(* Logix 5000 project; controller reports 1756-L63 rev 20.15; software revision 20.04; part 39 of 52 *)

        [72].log_data[43].total := -975.3802, [72].log_data[43].time := 3600.0, [72].log_data[43].valid := 1, [72].log_data[44].min := -0.30000305, [72].log_data[44].max := -0.30000305, [72].log_data[44].total := -1080.0911, [72].log_data[44].time := 3600.0, [72].log_data[44].valid := 1, [72].log_data[45].time := 3600.0, [72].log_data[45].valid := 1, [72].log_data[46].time := 3600.0, [72].log_data[46].valid := 1, [72].log_data[47].time := 3600.0, [72].log_data[47].valid := 1, [72].log_data[48].min := 6.57968, [72].log_data[48].max := 6.8025494, [72].log_data[48].total := 24189.488, [72].log_data[48].time := 3600.0, [72].log_data[48].minminute := 18, [72].log_data[48].maxminute := 33, [72].log_data[48].valid := 1, [72].log_data[49].min := 7.0676346, [72].log_data[49].max := 9.6694765, [72].log_data[49].total := 30225.078, [72].log_data[49].time := 3600.0, [72].log_data[49].minminute := 14, [72].log_data[49].maxminute := 59, [72].log_data[49].valid := 1, [72].log_data[50].min := 2.124167, [72].log_data[50].max := 2.2044892, [72].log_data[50].total := 7798.3384, [72].log_data[50].time := 3600.0, [72].log_data[50].minminute := 59, [72].log_data[50].maxminute := 1, [72].log_data[50].valid := 1, [72].log_data[51].time := 3600.0, [72].log_data[51].valid := 1, [72].log_data[52].min := -2.9800034, [72].log_data[52].max := 0.11999512, [72].log_data[52].total := -7899.8555, [72].log_data[52].time := 3600.0, [72].log_data[52].minminute := 36, [72].log_data[52].maxminute := 3, [72].log_data[52].valid := 1, [72].log_data[53].min := -2.5800018, [72].log_data[53].max := 0.19999695, [72].log_data[53].total := -7610.7764, [72].log_data[53].time := 3600.0, [72].log_data[53].minminute := 55, [72].log_data[53].maxminute := 9, [72].log_data[53].valid := 1, [72].log_data[54].max := 0.523, [72].log_data[54].total := 1217.2916, [72].log_data[54].time := 3600.0, [72].log_data[54].minminute := 3, [72].log_data[54].maxminute := 57, [72].log_data[54].valid := 1, [72].log_data[55].max := 0.509, [72].log_data[55].total := 1254.1338, [72].log_data[55].time := 3600.0,
        [72].log_data[55].minminute := 7, [72].log_data[55].maxminute := 9, [72].log_data[55].valid := 1, [72].log_data[56].min := 0.16004932, [72].log_data[56].max := 0.16055967, [72].log_data[56].total := 576.9628, [72].log_data[56].time := 3600.0, [72].log_data[56].minminute := 16, [72].log_data[56].maxminute := 29, [72].log_data[56].valid := 1, [72].log_data[57].min := 0.2558395, [72].log_data[57].max := 0.25772393, [72].log_data[57].total := 923.43195, [72].log_data[57].time := 3600.0, [72].log_data[57].minminute := 27, [72].log_data[57].maxminute := 4, [72].log_data[57].valid := 1, [72].log_data[58].time := 3600.0, [72].log_data[58].valid := 1, [72].log_data[59].time := 3600.0, [72].log_data[59].valid := 1, [72].log_data[60].valid := 1, [72].log_data[61].valid := 1, [72].log_data[62].valid := 1, [72].log_data[63].valid := 1, [72].log_data[64].valid := 1, [72].log_data[65].valid := 1, [72].log_data[66].valid := 1, [72].log_data[67].valid := 1, [72].log_data[68].valid := 1, [72].log_data[69].valid := 1, [72].log_data[70].valid := 1, [72].log_data[71].valid := 1, [72].log_data[72].valid := 1, [72].log_data[73].valid := 1, [72].log_data[74].valid := 1, [72].log_data[75].valid := 1, [72].log_data[76].valid := 1, [72].log_data[77].valid := 1, [72].log_data[78].valid := 1, [72].log_data[79].valid := 1, [72].log_data[80].valid := 1, [72].log_data[81].valid := 1, [72].log_data[82].valid := 1, [72].log_data[83].valid := 1, [72].log_data[84].valid := 1, [72].log_data[85].valid := 1, [72].log_data[86].valid := 1, [72].log_data[87].valid := 1, [72].log_data[88].valid := 1, [72].log_data[89].valid := 1, [72].log_data[90].valid := 1, [72].log_data[91].valid := 1, [72].log_data[92].valid := 1, [72].log_data[93].valid := 1, [72].log_data[94].valid := 1, [72].log_data[95].valid := 1, [72].log_data[96].valid := 1, [72].log_data[97].valid := 1, [72].log_data[98].valid := 1,
        [72].log_data[99].valid := 1, [72].log_data[100].valid := 1, [72].log_data[101].valid := 1, [72].log_data[102].valid := 1, [72].log_data[103].valid := 1, [72].log_data[104].valid := 1, [72].log_data[105].valid := 1, [72].log_data[106].valid := 1, [72].log_data[107].valid := 1, [72].log_data[108].valid := 1, [72].log_data[109].valid := 1, [72].log_data[110].valid := 1, [72].log_data[111].valid := 1, [72].log_data[112].valid := 1, [72].log_data[113].valid := 1, [72].log_data[114].valid := 1, [72].log_data[115].valid := 1, [72].log_data[116].valid := 1, [72].log_data[117].valid := 1, [72].log_data[118].valid := 1, [72].log_data[119].valid := 1, [72].log_data[120].valid := 1, [72].log_data[121].valid := 1, [72].log_data[122].valid := 1, [72].log_data[123].valid := 1, [72].log_data[124].valid := 1, [72].time.Year := 2023, [72].time.Month := 1, [72].time.Day := 16, [72].time.Hour := 3, [72].time.Minute := 59, [72].time.Second := 59, [73].log_data[0].min := 1.0, [73].log_data[0].max := 1.0, [73].log_data[0].total := 3600.0, [73].log_data[0].time := 3600.0, [73].log_data[0].valid := 1, [73].log_data[1].time := 3600.0, [73].log_data[1].valid := 1, [73].log_data[2].time := 3600.0, [73].log_data[2].valid := 1, [73].log_data[3].time := 3600.0, [73].log_data[3].valid := 1, [73].log_data[4].time := 3600.0, [73].log_data[4].valid := 1, [73].log_data[5].time := 3600.0, [73].log_data[5].valid := 1, [73].log_data[6].time := 3600.0, [73].log_data[6].valid := 1, [73].log_data[7].time := 3600.0, [73].log_data[7].valid := 1, [73].log_data[8].min := 1.0, [73].log_data[8].max := 1.0, [73].log_data[8].total := 3600.0, [73].log_data[8].time := 3600.0, [73].log_data[8].valid := 1, [73].log_data[9].min := 1.0, [73].log_data[9].max := 1.0, [73].log_data[9].total := 3600.0, [73].log_data[9].time := 3600.0,
        [73].log_data[9].valid := 1, [73].log_data[10].min := 1.0, [73].log_data[10].max := 1.0, [73].log_data[10].total := 3600.0, [73].log_data[10].time := 3600.0, [73].log_data[10].valid := 1, [73].log_data[11].time := 3600.0, [73].log_data[11].valid := 1, [73].log_data[12].min := 1.0, [73].log_data[12].max := 1.0, [73].log_data[12].total := 3600.0, [73].log_data[12].time := 3600.0, [73].log_data[12].valid := 1, [73].log_data[13].min := 1.0, [73].log_data[13].max := 1.0, [73].log_data[13].total := 3600.0, [73].log_data[13].time := 3600.0, [73].log_data[13].valid := 1, [73].log_data[14].time := 3600.0, [73].log_data[14].valid := 1, [73].log_data[15].time := 3600.0, [73].log_data[15].valid := 1, [73].log_data[16].time := 3600.0, [73].log_data[16].valid := 1, [73].log_data[17].min := 1.0, [73].log_data[17].max := 1.0, [73].log_data[17].total := 3600.0, [73].log_data[17].time := 3600.0, [73].log_data[17].valid := 1, [73].log_data[18].time := 3600.0, [73].log_data[18].valid := 1, [73].log_data[19].time := 3600.0, [73].log_data[19].valid := 1, [73].log_data[20].time := 3600.0, [73].log_data[20].valid := 1, [73].log_data[21].min := 1.0, [73].log_data[21].max := 1.0, [73].log_data[21].total := 3600.0, [73].log_data[21].time := 3600.0, [73].log_data[21].valid := 1, [73].log_data[22].time := 3600.0, [73].log_data[22].valid := 1, [73].log_data[23].time := 3600.0, [73].log_data[23].valid := 1, [73].log_data[24].time := 3600.0, [73].log_data[24].valid := 1, [73].log_data[25].time := 3600.0, [73].log_data[25].valid := 1, [73].log_data[26].time := 3600.0, [73].log_data[26].valid := 1, [73].log_data[27].time := 3600.0, [73].log_data[27].valid := 1, [73].log_data[28].time := 3600.0, [73].log_data[28].valid := 1, [73].log_data[29].min := 1.0, [73].log_data[29].max := 1.0, [73].log_data[29].total := 3600.0, [73].log_data[29].time := 3600.0, [73].log_data[29].valid := 1, [73].log_data[30].min := 1.0,
        [73].log_data[30].max := 1.0, [73].log_data[30].total := 3600.0, [73].log_data[30].time := 3600.0, [73].log_data[30].valid := 1, [73].log_data[31].max := 1.0, [73].log_data[31].total := 1498.749, [73].log_data[31].time := 3600.0, [73].log_data[31].minminute := 6, [73].log_data[31].valid := 1, [73].log_data[32].max := 1.0, [73].log_data[32].total := 1630.249, [73].log_data[32].time := 3600.0, [73].log_data[32].maxminute := 8, [73].log_data[32].valid := 1, [73].log_data[33].time := 3600.0, [73].log_data[33].valid := 1, [73].log_data[34].time := 3600.0, [73].log_data[34].valid := 1, [73].log_data[35].max := 1.0, [73].log_data[35].total := 1629.998, [73].log_data[35].time := 3600.0, [73].log_data[35].maxminute := 1, [73].log_data[35].valid := 1, [73].log_data[36].max := 1.0, [73].log_data[36].total := 1440.7471, [73].log_data[36].time := 3600.0, [73].log_data[36].valid := 1, [73].log_data[37].time := 3600.0, [73].log_data[37].valid := 1, [73].log_data[38].time := 3600.0, [73].log_data[38].valid := 1, [73].log_data[39].min := 0.99635506, [73].log_data[39].max := 1.0070726, [73].log_data[39].total := 3607.0815, [73].log_data[39].time := 3600.0, [73].log_data[39].minminute := 25, [73].log_data[39].maxminute := 53, [73].log_data[39].valid := 1, [73].log_data[40].min := 7.584652, [73].log_data[40].max := 7.597843, [73].log_data[40].total := 27334.826, [73].log_data[40].time := 3600.0, [73].log_data[40].minminute := 3, [73].log_data[40].maxminute := 12, [73].log_data[40].valid := 1, [73].log_data[41].min := 0.022540038, [73].log_data[41].max := 0.03529907, [73].log_data[41].total := 104.06682, [73].log_data[41].time := 3600.0, [73].log_data[41].maxminute := 33, [73].log_data[41].valid := 1, [73].log_data[42].min := 2.2918782, [73].log_data[42].max := 2.2964714, [73].log_data[42].total := 8259.474, [73].log_data[42].time := 3600.0, [73].log_data[42].minminute := 2, [73].log_data[42].maxminute := 2, [73].log_data[42].valid := 1, [73].log_data[43].min := -0.27999878, [73].log_data[43].max := -0.26000214,
        [73].log_data[43].total := -978.1933, [73].log_data[43].time := 3600.0, [73].log_data[43].valid := 1, [73].log_data[44].min := -0.30000305, [73].log_data[44].max := -0.30000305, [73].log_data[44].total := -1080.0911, [73].log_data[44].time := 3600.0, [73].log_data[44].valid := 1, [73].log_data[45].time := 3600.0, [73].log_data[45].valid := 1, [73].log_data[46].time := 3600.0, [73].log_data[46].valid := 1, [73].log_data[47].time := 3600.0, [73].log_data[47].valid := 1, [73].log_data[48].min := 6.747862, [73].log_data[48].max := 6.764351, [73].log_data[48].total := 24322.072, [73].log_data[48].time := 3600.0, [73].log_data[48].minminute := 58, [73].log_data[48].valid := 1, [73].log_data[49].min := 9.655932, [73].log_data[49].max := 9.74073, [73].log_data[49].total := 34957.934, [73].log_data[49].time := 3600.0, [73].log_data[49].maxminute := 58, [73].log_data[49].valid := 1, [73].log_data[50].min := 2.0386624, [73].log_data[50].max := 2.1277, [73].log_data[50].total := 7504.0176, [73].log_data[50].time := 3600.0, [73].log_data[50].minminute := 59, [73].log_data[50].valid := 1, [73].log_data[51].time := 3600.0, [73].log_data[51].valid := 1, [73].log_data[52].min := -3.1200027, [73].log_data[52].max := 0.11999512, [73].log_data[52].total := -8078.232, [73].log_data[52].time := 3600.0, [73].log_data[52].minminute := 18, [73].log_data[52].maxminute := 6, [73].log_data[52].valid := 1, [73].log_data[53].min := -2.6399994, [73].log_data[53].max := 0.16000366, [73].log_data[53].total := -7426.6094, [73].log_data[53].time := 3600.0, [73].log_data[53].minminute := 23, [73].log_data[53].maxminute := 1, [73].log_data[53].valid := 1, [73].log_data[54].max := 0.5445, [73].log_data[54].total := 1242.5043, [73].log_data[54].time := 3600.0, [73].log_data[54].minminute := 6, [73].log_data[54].maxminute := 18, [73].log_data[54].valid := 1, [73].log_data[55].max := 0.554, [73].log_data[55].total := 1217.1788, [73].log_data[55].time := 3600.0, [73].log_data[55].maxminute := 23, [73].log_data[55].valid := 1, [73].log_data[56].min := 0.16008857,
        [73].log_data[56].max := 0.16055967, [73].log_data[56].total := 576.96655, [73].log_data[56].time := 3600.0, [73].log_data[56].maxminute := 26, [73].log_data[56].valid := 1, [73].log_data[57].min := 0.255761, [73].log_data[57].max := 0.25619283, [73].log_data[57].total := 921.46454, [73].log_data[57].time := 3600.0, [73].log_data[57].minminute := 11, [73].log_data[57].maxminute := 14, [73].log_data[57].valid := 1, [73].log_data[58].time := 3600.0, [73].log_data[58].valid := 1, [73].log_data[59].time := 3600.0, [73].log_data[59].valid := 1, [73].log_data[60].valid := 1, [73].log_data[61].valid := 1, [73].log_data[62].valid := 1, [73].log_data[63].valid := 1, [73].log_data[64].valid := 1, [73].log_data[65].valid := 1, [73].log_data[66].valid := 1, [73].log_data[67].valid := 1, [73].log_data[68].valid := 1, [73].log_data[69].valid := 1, [73].log_data[70].valid := 1, [73].log_data[71].valid := 1, [73].log_data[72].valid := 1, [73].log_data[73].valid := 1, [73].log_data[74].valid := 1, [73].log_data[75].valid := 1, [73].log_data[76].valid := 1, [73].log_data[77].valid := 1, [73].log_data[78].valid := 1, [73].log_data[79].valid := 1, [73].log_data[80].valid := 1, [73].log_data[81].valid := 1, [73].log_data[82].valid := 1, [73].log_data[83].valid := 1, [73].log_data[84].valid := 1, [73].log_data[85].valid := 1, [73].log_data[86].valid := 1, [73].log_data[87].valid := 1, [73].log_data[88].valid := 1, [73].log_data[89].valid := 1, [73].log_data[90].valid := 1, [73].log_data[91].valid := 1, [73].log_data[92].valid := 1, [73].log_data[93].valid := 1, [73].log_data[94].valid := 1, [73].log_data[95].valid := 1, [73].log_data[96].valid := 1, [73].log_data[97].valid := 1, [73].log_data[98].valid := 1, [73].log_data[99].valid := 1, [73].log_data[100].valid := 1, [73].log_data[101].valid := 1, [73].log_data[102].valid := 1, [73].log_data[103].valid := 1,
        [73].log_data[104].valid := 1, [73].log_data[105].valid := 1, [73].log_data[106].valid := 1, [73].log_data[107].valid := 1, [73].log_data[108].valid := 1, [73].log_data[109].valid := 1, [73].log_data[110].valid := 1, [73].log_data[111].valid := 1, [73].log_data[112].valid := 1, [73].log_data[113].valid := 1, [73].log_data[114].valid := 1, [73].log_data[115].valid := 1, [73].log_data[116].valid := 1, [73].log_data[117].valid := 1, [73].log_data[118].valid := 1, [73].log_data[119].valid := 1, [73].log_data[120].valid := 1, [73].log_data[121].valid := 1, [73].log_data[122].valid := 1, [73].log_data[123].valid := 1, [73].log_data[124].valid := 1, [73].time.Year := 2023, [73].time.Month := 1, [73].time.Day := 16, [73].time.Hour := 4, [73].time.Minute := 59, [73].time.Second := 59, [74].log_data[0].min := 1.0, [74].log_data[0].max := 1.0, [74].log_data[0].total := 3600.0, [74].log_data[0].time := 3600.0, [74].log_data[0].valid := 1, [74].log_data[1].time := 3600.0, [74].log_data[1].valid := 1, [74].log_data[2].time := 3600.0, [74].log_data[2].valid := 1, [74].log_data[3].time := 3600.0, [74].log_data[3].valid := 1, [74].log_data[4].time := 3600.0, [74].log_data[4].valid := 1, [74].log_data[5].time := 3600.0, [74].log_data[5].valid := 1, [74].log_data[6].time := 3600.0, [74].log_data[6].valid := 1, [74].log_data[7].time := 3600.0, [74].log_data[7].valid := 1, [74].log_data[8].max := 1.0, [74].log_data[8].total := 1742.751, [74].log_data[8].time := 3600.0, [74].log_data[8].minminute := 29, [74].log_data[8].valid := 1, [74].log_data[9].max := 1.0, [74].log_data[9].total := 1742.751, [74].log_data[9].time := 3600.0, [74].log_data[9].minminute := 29, [74].log_data[9].valid := 1, [74].log_data[10].min := 1.0, [74].log_data[10].max := 1.0, [74].log_data[10].total := 3600.0, [74].log_data[10].time := 3600.0,
        [74].log_data[10].valid := 1, [74].log_data[11].time := 3600.0, [74].log_data[11].valid := 1, [74].log_data[12].min := 1.0, [74].log_data[12].max := 1.0, [74].log_data[12].total := 3600.0, [74].log_data[12].time := 3600.0, [74].log_data[12].valid := 1, [74].log_data[13].min := 1.0, [74].log_data[13].max := 1.0, [74].log_data[13].total := 3600.0, [74].log_data[13].time := 3600.0, [74].log_data[13].valid := 1, [74].log_data[14].time := 3600.0, [74].log_data[14].valid := 1, [74].log_data[15].time := 3600.0, [74].log_data[15].valid := 1, [74].log_data[16].time := 3600.0, [74].log_data[16].valid := 1, [74].log_data[17].min := 1.0, [74].log_data[17].max := 1.0, [74].log_data[17].total := 3600.0, [74].log_data[17].time := 3600.0, [74].log_data[17].valid := 1, [74].log_data[18].time := 3600.0, [74].log_data[18].valid := 1, [74].log_data[19].time := 3600.0, [74].log_data[19].valid := 1, [74].log_data[20].time := 3600.0, [74].log_data[20].valid := 1, [74].log_data[21].min := 1.0, [74].log_data[21].max := 1.0, [74].log_data[21].total := 3600.0, [74].log_data[21].time := 3600.0, [74].log_data[21].valid := 1, [74].log_data[22].time := 3600.0, [74].log_data[22].valid := 1, [74].log_data[23].time := 3600.0, [74].log_data[23].valid := 1, [74].log_data[24].time := 3600.0, [74].log_data[24].valid := 1, [74].log_data[25].time := 3600.0, [74].log_data[25].valid := 1, [74].log_data[26].time := 3600.0, [74].log_data[26].valid := 1, [74].log_data[27].time := 3600.0, [74].log_data[27].valid := 1, [74].log_data[28].time := 3600.0, [74].log_data[28].valid := 1, [74].log_data[29].min := 1.0, [74].log_data[29].max := 1.0, [74].log_data[29].total := 3600.0, [74].log_data[29].time := 3600.0, [74].log_data[29].valid := 1, [74].log_data[30].min := 1.0, [74].log_data[30].max := 1.0, [74].log_data[30].total := 3600.0, [74].log_data[30].time := 3600.0, [74].log_data[30].valid := 1, [74].log_data[31].max := 1.0,
        [74].log_data[31].total := 968.99805, [74].log_data[31].time := 3600.0, [74].log_data[31].valid := 1, [74].log_data[32].max := 1.0, [74].log_data[32].total := 543.249, [74].log_data[32].time := 3600.0, [74].log_data[32].maxminute := 11, [74].log_data[32].valid := 1, [74].log_data[33].time := 3600.0, [74].log_data[33].valid := 1, [74].log_data[34].time := 3600.0, [74].log_data[34].valid := 1, [74].log_data[35].max := 1.0, [74].log_data[35].total := 724.749, [74].log_data[35].time := 3600.0, [74].log_data[35].maxminute := 5, [74].log_data[35].valid := 1, [74].log_data[36].max := 1.0, [74].log_data[36].total := 756.749, [74].log_data[36].time := 3600.0, [74].log_data[36].minminute := 3, [74].log_data[36].valid := 1, [74].log_data[37].time := 3600.0, [74].log_data[37].valid := 1, [74].log_data[38].time := 3600.0, [74].log_data[38].valid := 1, [74].log_data[39].min := 0.9936463, [74].log_data[39].max := 1.0061305, [74].log_data[39].total := 3601.6323, [74].log_data[39].time := 3600.0, [74].log_data[39].minminute := 3, [74].log_data[39].valid := 1, [74].log_data[40].min := 7.561569, [74].log_data[40].max := 7.609111, [74].log_data[40].total := 27332.018, [74].log_data[40].time := 3600.0, [74].log_data[40].minminute := 2, [74].log_data[40].maxminute := 4, [74].log_data[40].valid := 1, [74].log_data[41].min := 0.022540038, [74].log_data[41].max := 0.033139892, [74].log_data[41].total := 93.51873, [74].log_data[41].time := 3600.0, [74].log_data[41].minminute := 16, [74].log_data[41].valid := 1, [74].log_data[42].min := 2.2917604, [74].log_data[42].max := 2.2964714, [74].log_data[42].total := 8259.399, [74].log_data[42].time := 3600.0, [74].log_data[42].minminute := 17, [74].log_data[42].maxminute := 59, [74].log_data[42].valid := 1, [74].log_data[43].min := -0.27999878, [74].log_data[43].max := -0.26000214, [74].log_data[43].total := -968.6149, [74].log_data[43].time := 3600.0, [74].log_data[43].valid := 1, [74].log_data[44].min := -0.30000305, [74].log_data[44].max := -0.27999878, [74].log_data[44].total := -1080.0759,
        [74].log_data[44].time := 3600.0, [74].log_data[44].maxminute := 46, [74].log_data[44].valid := 1, [74].log_data[45].time := 3600.0, [74].log_data[45].valid := 1, [74].log_data[46].time := 3600.0, [74].log_data[46].valid := 1, [74].log_data[47].time := 3600.0, [74].log_data[47].valid := 1, [74].log_data[48].min := 6.734946, [74].log_data[48].max := 6.750061, [74].log_data[48].total := 24266.814, [74].log_data[48].time := 3600.0, [74].log_data[48].minminute := 35, [74].log_data[48].valid := 1, [74].log_data[49].min := 9.64867, [74].log_data[49].max := 9.741908, [74].log_data[49].total := 34884.496, [74].log_data[49].time := 3600.0, [74].log_data[49].minminute := 44, [74].log_data[49].maxminute := 8, [74].log_data[49].valid := 1, [74].log_data[50].min := 1.9993255, [74].log_data[50].max := 2.1042628, [74].log_data[50].total := 7410.9795, [74].log_data[50].time := 3600.0, [74].log_data[50].minminute := 29, [74].log_data[50].maxminute := 53, [74].log_data[50].valid := 1, [74].log_data[51].time := 3600.0, [74].log_data[51].valid := 1, [74].log_data[52].min := -3.0800018, [74].log_data[52].max := 0.11999512, [74].log_data[52].total := -6464.315, [74].log_data[52].time := 3600.0, [74].log_data[52].minminute := 1, [74].log_data[52].valid := 1, [74].log_data[53].min := -2.5800018, [74].log_data[53].max := 0.19999695, [74].log_data[53].total := -5924.441, [74].log_data[53].time := 3600.0, [74].log_data[53].minminute := 16, [74].log_data[53].maxminute := 4, [74].log_data[53].valid := 1, [74].log_data[54].max := 0.55050004, [74].log_data[54].total := 599.9697, [74].log_data[54].time := 3600.0, [74].log_data[54].maxminute := 22, [74].log_data[54].valid := 1, [74].log_data[55].max := 0.5245, [74].log_data[55].total := 587.57196, [74].log_data[55].time := 3600.0, [74].log_data[55].minminute := 3, [74].log_data[55].maxminute := 26, [74].log_data[55].valid := 1, [74].log_data[56].min := 0.16004932, [74].log_data[56].max := 0.16055967, [74].log_data[56].total := 576.99097, [74].log_data[56].time := 3600.0, [74].log_data[56].minminute := 23,
        [74].log_data[56].maxminute := 52, [74].log_data[56].valid := 1, [74].log_data[57].min := 0.25580025, [74].log_data[57].max := 0.25619283, [74].log_data[57].total := 921.4573, [74].log_data[57].time := 3600.0, [74].log_data[57].minminute := 4, [74].log_data[57].maxminute := 11, [74].log_data[57].valid := 1, [74].log_data[58].time := 3600.0, [74].log_data[58].valid := 1, [74].log_data[59].time := 3600.0, [74].log_data[59].valid := 1, [74].log_data[60].valid := 1, [74].log_data[61].valid := 1, [74].log_data[62].valid := 1, [74].log_data[63].valid := 1, [74].log_data[64].valid := 1, [74].log_data[65].valid := 1, [74].log_data[66].valid := 1, [74].log_data[67].valid := 1, [74].log_data[68].valid := 1, [74].log_data[69].valid := 1, [74].log_data[70].valid := 1, [74].log_data[71].valid := 1, [74].log_data[72].valid := 1, [74].log_data[73].valid := 1, [74].log_data[74].valid := 1, [74].log_data[75].valid := 1, [74].log_data[76].valid := 1, [74].log_data[77].valid := 1, [74].log_data[78].valid := 1, [74].log_data[79].valid := 1, [74].log_data[80].valid := 1, [74].log_data[81].valid := 1, [74].log_data[82].valid := 1, [74].log_data[83].valid := 1, [74].log_data[84].valid := 1, [74].log_data[85].valid := 1, [74].log_data[86].valid := 1, [74].log_data[87].valid := 1, [74].log_data[88].valid := 1, [74].log_data[89].valid := 1, [74].log_data[90].valid := 1, [74].log_data[91].valid := 1, [74].log_data[92].valid := 1, [74].log_data[93].valid := 1, [74].log_data[94].valid := 1, [74].log_data[95].valid := 1, [74].log_data[96].valid := 1, [74].log_data[97].valid := 1, [74].log_data[98].valid := 1, [74].log_data[99].valid := 1, [74].log_data[100].valid := 1, [74].log_data[101].valid := 1, [74].log_data[102].valid := 1, [74].log_data[103].valid := 1, [74].log_data[104].valid := 1, [74].log_data[105].valid := 1, [74].log_data[106].valid := 1,
        [74].log_data[107].valid := 1, [74].log_data[108].valid := 1, [74].log_data[109].valid := 1, [74].log_data[110].valid := 1, [74].log_data[111].valid := 1, [74].log_data[112].valid := 1, [74].log_data[113].valid := 1, [74].log_data[114].valid := 1, [74].log_data[115].valid := 1, [74].log_data[116].valid := 1, [74].log_data[117].valid := 1, [74].log_data[118].valid := 1, [74].log_data[119].valid := 1, [74].log_data[120].valid := 1, [74].log_data[121].valid := 1, [74].log_data[122].valid := 1, [74].log_data[123].valid := 1, [74].log_data[124].valid := 1, [74].time.Year := 2023, [74].time.Month := 1, [74].time.Day := 16, [74].time.Hour := 5, [74].time.Minute := 59, [74].time.Second := 59, [75].log_data[0].min := 1.0, [75].log_data[0].max := 1.0, [75].log_data[0].total := 3600.0, [75].log_data[0].time := 3600.0, [75].log_data[0].valid := 1, [75].log_data[1].time := 3600.0, [75].log_data[1].valid := 1, [75].log_data[2].time := 3600.0, [75].log_data[2].valid := 1, [75].log_data[3].time := 3600.0, [75].log_data[3].valid := 1, [75].log_data[4].time := 3600.0, [75].log_data[4].valid := 1, [75].log_data[5].time := 3600.0, [75].log_data[5].valid := 1, [75].log_data[6].time := 3600.0, [75].log_data[6].valid := 1, [75].log_data[7].time := 3600.0, [75].log_data[7].valid := 1, [75].log_data[8].time := 3600.0, [75].log_data[8].valid := 1, [75].log_data[9].time := 3600.0, [75].log_data[9].valid := 1, [75].log_data[10].min := 1.0, [75].log_data[10].max := 1.0, [75].log_data[10].total := 3600.0, [75].log_data[10].time := 3600.0, [75].log_data[10].valid := 1, [75].log_data[11].time := 3600.0, [75].log_data[11].valid := 1, [75].log_data[12].min := 1.0, [75].log_data[12].max := 1.0, [75].log_data[12].total := 3600.0, [75].log_data[12].time := 3600.0, [75].log_data[12].valid := 1, [75].log_data[13].min := 1.0,
        [75].log_data[13].max := 1.0, [75].log_data[13].total := 3600.0, [75].log_data[13].time := 3600.0, [75].log_data[13].valid := 1, [75].log_data[14].time := 3600.0, [75].log_data[14].valid := 1, [75].log_data[15].time := 3600.0, [75].log_data[15].valid := 1, [75].log_data[16].time := 3600.0, [75].log_data[16].valid := 1, [75].log_data[17].min := 1.0, [75].log_data[17].max := 1.0, [75].log_data[17].total := 3600.0, [75].log_data[17].time := 3600.0, [75].log_data[17].valid := 1, [75].log_data[18].time := 3600.0, [75].log_data[18].valid := 1, [75].log_data[19].time := 3600.0, [75].log_data[19].valid := 1, [75].log_data[20].time := 3600.0, [75].log_data[20].valid := 1, [75].log_data[21].min := 1.0, [75].log_data[21].max := 1.0, [75].log_data[21].total := 3600.0, [75].log_data[21].time := 3600.0, [75].log_data[21].valid := 1, [75].log_data[22].time := 3600.0, [75].log_data[22].valid := 1, [75].log_data[23].time := 3600.0, [75].log_data[23].valid := 1, [75].log_data[24].time := 3600.0, [75].log_data[24].valid := 1, [75].log_data[25].time := 3600.0, [75].log_data[25].valid := 1, [75].log_data[26].time := 3600.0, [75].log_data[26].valid := 1, [75].log_data[27].time := 3600.0, [75].log_data[27].valid := 1, [75].log_data[28].time := 3600.0, [75].log_data[28].valid := 1, [75].log_data[29].min := 1.0, [75].log_data[29].max := 1.0, [75].log_data[29].total := 3600.0, [75].log_data[29].time := 3600.0, [75].log_data[29].valid := 1, [75].log_data[30].min := 1.0, [75].log_data[30].max := 1.0, [75].log_data[30].total := 3600.0, [75].log_data[30].time := 3600.0, [75].log_data[30].valid := 1, [75].log_data[31].time := 3600.0, [75].log_data[31].valid := 1, [75].log_data[32].time := 3600.0, [75].log_data[32].valid := 1, [75].log_data[33].time := 3600.0, [75].log_data[33].valid := 1, [75].log_data[34].time := 3600.0, [75].log_data[34].valid := 1, [75].log_data[35].time := 3600.0, [75].log_data[35].valid := 1,
        [75].log_data[36].time := 3600.0, [75].log_data[36].valid := 1, [75].log_data[37].time := 3600.0, [75].log_data[37].valid := 1, [75].log_data[38].time := 3600.0, [75].log_data[38].valid := 1, [75].log_data[39].min := 0.9941174, [75].log_data[39].max := 1.0055416, [75].log_data[39].total := 3601.261, [75].log_data[39].time := 3600.0, [75].log_data[39].minminute := 36, [75].log_data[39].maxminute := 43, [75].log_data[39].valid := 1, [75].log_data[40].min := 7.574485, [75].log_data[40].max := 7.6107597, [75].log_data[40].total := 27331.771, [75].log_data[40].time := 3600.0, [75].log_data[40].minminute := 34, [75].log_data[40].maxminute := 32, [75].log_data[40].valid := 1, [75].log_data[41].min := 0.022540038, [75].log_data[41].max := 0.039224852, [75].log_data[41].total := 90.41001, [75].log_data[41].time := 3600.0, [75].log_data[41].maxminute := 5, [75].log_data[41].valid := 1, [75].log_data[42].min := 2.2917604, [75].log_data[42].max := 2.2963536, [75].log_data[42].total := 8259.333, [75].log_data[42].time := 3600.0, [75].log_data[42].minminute := 3, [75].log_data[42].maxminute := 10, [75].log_data[42].valid := 1, [75].log_data[43].min := -0.27999878, [75].log_data[43].max := -0.26000214, [75].log_data[43].total := -959.8148, [75].log_data[43].time := 3600.0, [75].log_data[43].valid := 1, [75].log_data[44].min := -0.30000305, [75].log_data[44].max := -0.30000305, [75].log_data[44].total := -1080.0911, [75].log_data[44].time := 3600.0, [75].log_data[44].valid := 1, [75].log_data[45].time := 3600.0, [75].log_data[45].valid := 1, [75].log_data[46].time := 3600.0, [75].log_data[46].valid := 1, [75].log_data[47].time := 3600.0, [75].log_data[47].valid := 1, [75].log_data[48].min := 6.7382436, [75].log_data[48].max := 6.7473125, [75].log_data[48].total := 24275.645, [75].log_data[48].time := 3600.0, [75].log_data[48].maxminute := 48, [75].log_data[48].valid := 1, [75].log_data[49].min := 9.64553, [75].log_data[49].max := 9.706968, [75].log_data[49].total := 34838.707, [75].log_data[49].time := 3600.0, [75].log_data[49].minminute := 5,
        [75].log_data[49].maxminute := 48, [75].log_data[49].valid := 1, [75].log_data[50].min := 2.0994341, [75].log_data[50].max := 2.1086206, [75].log_data[50].total := 7579.887, [75].log_data[50].time := 3600.0, [75].log_data[50].maxminute := 44, [75].log_data[50].valid := 1, [75].log_data[51].time := 3600.0, [75].log_data[51].valid := 1, [75].log_data[52].min := -1.5999985, [75].log_data[52].max := -1.4400024, [75].log_data[52].total := -5502.215, [75].log_data[52].time := 3600.0, [75].log_data[52].minminute := 51, [75].log_data[52].maxminute := 15, [75].log_data[52].valid := 1, [75].log_data[53].min := -1.4400024, [75].log_data[53].max := -1.2399979, [75].log_data[53].total := -4781.3306, [75].log_data[53].time := 3600.0, [75].log_data[53].minminute := 7, [75].log_data[53].maxminute := 54, [75].log_data[53].valid := 1, [75].log_data[54].time := 3600.0, [75].log_data[54].valid := 1, [75].log_data[55].time := 3600.0, [75].log_data[55].valid := 1, [75].log_data[56].min := 0.16004932, [75].log_data[56].max := 0.16055967, [75].log_data[56].total := 576.94586, [75].log_data[56].time := 3600.0, [75].log_data[56].minminute := 8, [75].log_data[56].maxminute := 13, [75].log_data[56].valid := 1, [75].log_data[57].min := 0.25580025, [75].log_data[57].max := 0.25627133, [75].log_data[57].total := 921.7233, [75].log_data[57].time := 3600.0, [75].log_data[57].minminute := 24, [75].log_data[57].maxminute := 32, [75].log_data[57].valid := 1, [75].log_data[58].time := 3600.0, [75].log_data[58].valid := 1, [75].log_data[59].time := 3600.0, [75].log_data[59].valid := 1, [75].log_data[60].valid := 1, [75].log_data[61].valid := 1, [75].log_data[62].valid := 1, [75].log_data[63].valid := 1, [75].log_data[64].valid := 1, [75].log_data[65].valid := 1, [75].log_data[66].valid := 1, [75].log_data[67].valid := 1, [75].log_data[68].valid := 1, [75].log_data[69].valid := 1, [75].log_data[70].valid := 1, [75].log_data[71].valid := 1, [75].log_data[72].valid := 1, [75].log_data[73].valid := 1,
        [75].log_data[74].valid := 1, [75].log_data[75].valid := 1, [75].log_data[76].valid := 1, [75].log_data[77].valid := 1, [75].log_data[78].valid := 1, [75].log_data[79].valid := 1, [75].log_data[80].valid := 1, [75].log_data[81].valid := 1, [75].log_data[82].valid := 1, [75].log_data[83].valid := 1, [75].log_data[84].valid := 1, [75].log_data[85].valid := 1, [75].log_data[86].valid := 1, [75].log_data[87].valid := 1, [75].log_data[88].valid := 1, [75].log_data[89].valid := 1, [75].log_data[90].valid := 1, [75].log_data[91].valid := 1, [75].log_data[92].valid := 1, [75].log_data[93].valid := 1, [75].log_data[94].valid := 1, [75].log_data[95].valid := 1, [75].log_data[96].valid := 1, [75].log_data[97].valid := 1, [75].log_data[98].valid := 1, [75].log_data[99].valid := 1, [75].log_data[100].valid := 1, [75].log_data[101].valid := 1, [75].log_data[102].valid := 1, [75].log_data[103].valid := 1, [75].log_data[104].valid := 1, [75].log_data[105].valid := 1, [75].log_data[106].valid := 1, [75].log_data[107].valid := 1, [75].log_data[108].valid := 1, [75].log_data[109].valid := 1, [75].log_data[110].valid := 1, [75].log_data[111].valid := 1, [75].log_data[112].valid := 1, [75].log_data[113].valid := 1, [75].log_data[114].valid := 1, [75].log_data[115].valid := 1, [75].log_data[116].valid := 1, [75].log_data[117].valid := 1, [75].log_data[118].valid := 1, [75].log_data[119].valid := 1, [75].log_data[120].valid := 1, [75].log_data[121].valid := 1, [75].log_data[122].valid := 1, [75].log_data[123].valid := 1, [75].log_data[124].valid := 1, [75].time.Year := 2023, [75].time.Month := 1, [75].time.Day := 16, [75].time.Hour := 6, [75].time.Minute := 59, [75].time.Second := 59, [76].log_data[0].min := 1.0, [76].log_data[0].max := 1.0, [76].log_data[0].total := 3600.0,
        [76].log_data[0].time := 3600.0, [76].log_data[0].valid := 1, [76].log_data[1].max := 1.0, [76].log_data[1].total := 546.5, [76].log_data[1].time := 3600.0, [76].log_data[1].maxminute := 36, [76].log_data[1].valid := 1, [76].log_data[2].max := 1.0, [76].log_data[2].total := 543.0, [76].log_data[2].time := 3600.0, [76].log_data[2].maxminute := 36, [76].log_data[2].valid := 1, [76].log_data[3].time := 3600.0, [76].log_data[3].valid := 1, [76].log_data[4].time := 3600.0, [76].log_data[4].valid := 1, [76].log_data[5].max := 1.0, [76].log_data[5].total := 227.5, [76].log_data[5].time := 3600.0, [76].log_data[5].maxminute := 38, [76].log_data[5].valid := 1, [76].log_data[6].time := 3600.0, [76].log_data[6].valid := 1, [76].log_data[7].time := 3600.0, [76].log_data[7].valid := 1, [76].log_data[8].max := 1.0, [76].log_data[8].total := 1171.249, [76].log_data[8].time := 3600.0, [76].log_data[8].maxminute := 40, [76].log_data[8].valid := 1, [76].log_data[9].max := 1.0, [76].log_data[9].total := 1167.749, [76].log_data[9].time := 3600.0, [76].log_data[9].maxminute := 40, [76].log_data[9].valid := 1, [76].log_data[10].min := 1.0, [76].log_data[10].max := 1.0, [76].log_data[10].total := 3600.0, [76].log_data[10].time := 3600.0, [76].log_data[10].valid := 1, [76].log_data[11].time := 3600.0, [76].log_data[11].valid := 1, [76].log_data[12].min := 1.0, [76].log_data[12].max := 1.0, [76].log_data[12].total := 3600.0, [76].log_data[12].time := 3600.0, [76].log_data[12].valid := 1, [76].log_data[13].min := 1.0, [76].log_data[13].max := 1.0, [76].log_data[13].total := 3600.0, [76].log_data[13].time := 3600.0, [76].log_data[13].valid := 1, [76].log_data[14].time := 3600.0, [76].log_data[14].valid := 1, [76].log_data[15].time := 3600.0, [76].log_data[15].valid := 1, [76].log_data[16].time := 3600.0, [76].log_data[16].valid := 1, [76].log_data[17].min := 1.0, [76].log_data[17].max := 1.0,
        [76].log_data[17].total := 3600.0, [76].log_data[17].time := 3600.0, [76].log_data[17].valid := 1, [76].log_data[18].time := 3600.0, [76].log_data[18].valid := 1, [76].log_data[19].time := 3600.0, [76].log_data[19].valid := 1, [76].log_data[20].time := 3600.0, [76].log_data[20].valid := 1, [76].log_data[21].min := 1.0, [76].log_data[21].max := 1.0, [76].log_data[21].total := 3600.0, [76].log_data[21].time := 3600.0, [76].log_data[21].valid := 1, [76].log_data[22].time := 3600.0, [76].log_data[22].valid := 1, [76].log_data[23].time := 3600.0, [76].log_data[23].valid := 1, [76].log_data[24].time := 3600.0, [76].log_data[24].valid := 1, [76].log_data[25].time := 3600.0, [76].log_data[25].valid := 1, [76].log_data[26].time := 3600.0, [76].log_data[26].valid := 1, [76].log_data[27].time := 3600.0, [76].log_data[27].valid := 1, [76].log_data[28].time := 3600.0, [76].log_data[28].valid := 1, [76].log_data[29].min := 1.0, [76].log_data[29].max := 1.0, [76].log_data[29].total := 3600.0, [76].log_data[29].time := 3600.0, [76].log_data[29].valid := 1, [76].log_data[30].min := 1.0, [76].log_data[30].max := 1.0, [76].log_data[30].total := 3600.0, [76].log_data[30].time := 3600.0, [76].log_data[30].valid := 1, [76].log_data[31].max := 1.0, [76].log_data[31].total := 543.249, [76].log_data[31].time := 3600.0, [76].log_data[31].maxminute := 44, [76].log_data[31].valid := 1, [76].log_data[32].max := 1.0, [76].log_data[32].total := 444.498, [76].log_data[32].time := 3600.0, [76].log_data[32].maxminute := 40, [76].log_data[32].valid := 1, [76].log_data[33].time := 3600.0, [76].log_data[33].valid := 1, [76].log_data[34].time := 3600.0, [76].log_data[34].valid := 1, [76].log_data[35].max := 1.0, [76].log_data[35].total := 543.249, [76].log_data[35].time := 3600.0, [76].log_data[35].maxminute := 48, [76].log_data[35].valid := 1, [76].log_data[36].max := 1.0, [76].log_data[36].total := 440.998, [76].log_data[36].time := 3600.0,
        [76].log_data[36].maxminute := 40, [76].log_data[36].valid := 1, [76].log_data[37].max := 7.3416233, [76].log_data[37].total := 3478.435, [76].log_data[37].time := 3600.0, [76].log_data[37].maxminute := 38, [76].log_data[37].valid := 1, [76].log_data[38].time := 3600.0, [76].log_data[38].valid := 1, [76].log_data[39].min := 0.99435294, [76].log_data[39].max := 1.0215589, [76].log_data[39].total := 3607.7969, [76].log_data[39].time := 3600.0, [76].log_data[39].minminute := 14, [76].log_data[39].maxminute := 43, [76].log_data[39].valid := 1, [76].log_data[40].min := 7.584652, [76].log_data[40].max := 7.6019654, [76].log_data[40].total := 27338.77, [76].log_data[40].time := 3600.0, [76].log_data[40].minminute := 29, [76].log_data[40].maxminute := 5, [76].log_data[40].valid := 1, [76].log_data[41].min := 0.022540038, [76].log_data[41].max := 0.037261963, [76].log_data[41].total := 114.78345, [76].log_data[41].time := 3600.0, [76].log_data[41].maxminute := 41, [76].log_data[41].valid := 1, [76].log_data[42].min := 2.2917604, [76].log_data[42].max := 2.2964714, [76].log_data[42].total := 8259.297, [76].log_data[42].time := 3600.0, [76].log_data[42].minminute := 52, [76].log_data[42].maxminute := 20, [76].log_data[42].valid := 1, [76].log_data[43].min := -0.27999878, [76].log_data[43].max := -0.26000214, [76].log_data[43].total := -980.99854, [76].log_data[43].time := 3600.0, [76].log_data[43].valid := 1, [76].log_data[44].min := -0.30000305, [76].log_data[44].max := -0.30000305, [76].log_data[44].total := -1080.0911, [76].log_data[44].time := 3600.0, [76].log_data[44].valid := 1, [76].log_data[45].time := 3600.0, [76].log_data[45].valid := 1, [76].log_data[46].time := 3600.0, [76].log_data[46].valid := 1, [76].log_data[47].time := 3600.0, [76].log_data[47].valid := 1, [76].log_data[48].min := 6.6335416, [76].log_data[48].max := 6.9465485, [76].log_data[48].total := 24319.84, [76].log_data[48].time := 3600.0, [76].log_data[48].minminute := 59, [76].log_data[48].maxminute := 45, [76].log_data[48].valid := 1, [76].log_data[49].min := 7.204253,
        [76].log_data[49].max := 9.739357, [76].log_data[49].total := 33188.277, [76].log_data[49].time := 3600.0, [76].log_data[49].minminute := 59, [76].log_data[49].maxminute := 28, [76].log_data[49].valid := 1, [76].log_data[50].min := 2.061864, [76].log_data[50].max := 2.1505485, [76].log_data[50].total := 7572.1, [76].log_data[50].time := 3600.0, [76].log_data[50].minminute := 43, [76].log_data[50].maxminute := 40, [76].log_data[50].valid := 1, [76].log_data[51].time := 3600.0, [76].log_data[51].valid := 1, [76].log_data[52].min := -4.199997, [76].log_data[52].max := 0.11999512, [76].log_data[52].total := -6285.726, [76].log_data[52].time := 3600.0, [76].log_data[52].minminute := 40, [76].log_data[52].maxminute := 42, [76].log_data[52].valid := 1, [76].log_data[53].min := -3.9399948, [76].log_data[53].max := 0.27999878, [76].log_data[53].total := -5460.3057, [76].log_data[53].time := 3600.0, [76].log_data[53].minminute := 40, [76].log_data[53].maxminute := 58, [76].log_data[53].valid := 1, [76].log_data[54].max := 0.5535, [76].log_data[54].total := 389.23734, [76].log_data[54].time := 3600.0, [76].log_data[54].maxminute := 54, [76].log_data[54].valid := 1, [76].log_data[55].max := 0.5175, [76].log_data[55].total := 387.67783, [76].log_data[55].time := 3600.0, [76].log_data[55].maxminute := 40, [76].log_data[55].valid := 1, [76].log_data[56].min := 0.16008857, [76].log_data[56].max := 0.16048115, [76].log_data[56].total := 576.83215, [76].log_data[56].time := 3600.0, [76].log_data[56].minminute := 40, [76].log_data[56].maxminute := 14, [76].log_data[56].valid := 1, [76].log_data[57].min := 0.2558395, [76].log_data[57].max := 0.25627133, [76].log_data[57].total := 921.702, [76].log_data[57].time := 3600.0, [76].log_data[57].minminute := 41, [76].log_data[57].valid := 1, [76].log_data[58].time := 3600.0, [76].log_data[58].valid := 1, [76].log_data[59].time := 3600.0, [76].log_data[59].valid := 1, [76].log_data[60].valid := 1, [76].log_data[61].valid := 1, [76].log_data[62].valid := 1, [76].log_data[63].valid := 1,
        [76].log_data[64].valid := 1, [76].log_data[65].valid := 1, [76].log_data[66].valid := 1, [76].log_data[67].valid := 1, [76].log_data[68].valid := 1, [76].log_data[69].valid := 1, [76].log_data[70].valid := 1, [76].log_data[71].valid := 1, [76].log_data[72].valid := 1, [76].log_data[73].valid := 1, [76].log_data[74].valid := 1, [76].log_data[75].valid := 1, [76].log_data[76].valid := 1, [76].log_data[77].valid := 1, [76].log_data[78].valid := 1, [76].log_data[79].valid := 1, [76].log_data[80].valid := 1, [76].log_data[81].valid := 1, [76].log_data[82].valid := 1, [76].log_data[83].valid := 1, [76].log_data[84].valid := 1, [76].log_data[85].valid := 1, [76].log_data[86].valid := 1, [76].log_data[87].valid := 1, [76].log_data[88].valid := 1, [76].log_data[89].valid := 1, [76].log_data[90].valid := 1, [76].log_data[91].valid := 1, [76].log_data[92].valid := 1, [76].log_data[93].valid := 1, [76].log_data[94].valid := 1, [76].log_data[95].valid := 1, [76].log_data[96].valid := 1, [76].log_data[97].valid := 1, [76].log_data[98].valid := 1, [76].log_data[99].valid := 1, [76].log_data[100].valid := 1, [76].log_data[101].valid := 1, [76].log_data[102].valid := 1, [76].log_data[103].valid := 1, [76].log_data[104].valid := 1, [76].log_data[105].valid := 1, [76].log_data[106].valid := 1, [76].log_data[107].valid := 1, [76].log_data[108].valid := 1, [76].log_data[109].valid := 1, [76].log_data[110].valid := 1, [76].log_data[111].valid := 1, [76].log_data[112].valid := 1, [76].log_data[113].valid := 1, [76].log_data[114].valid := 1, [76].log_data[115].valid := 1, [76].log_data[116].valid := 1, [76].log_data[117].valid := 1, [76].log_data[118].valid := 1, [76].log_data[119].valid := 1, [76].log_data[120].valid := 1, [76].log_data[121].valid := 1, [76].log_data[122].valid := 1, [76].log_data[123].valid := 1,
        [76].log_data[124].valid := 1, [76].time.Year := 2023, [76].time.Month := 1, [76].time.Day := 16, [76].time.Hour := 7, [76].time.Minute := 59, [76].time.Second := 59, [77].log_data[0].min := 1.0, [77].log_data[0].max := 1.0, [77].log_data[0].total := 3600.0, [77].log_data[0].time := 3600.0, [77].log_data[0].valid := 1, [77].log_data[1].time := 3600.0, [77].log_data[1].valid := 1, [77].log_data[2].time := 3600.0, [77].log_data[2].valid := 1, [77].log_data[3].time := 3600.0, [77].log_data[3].valid := 1, [77].log_data[4].time := 3600.0, [77].log_data[4].valid := 1, [77].log_data[5].time := 3600.0, [77].log_data[5].valid := 1, [77].log_data[6].time := 3600.0, [77].log_data[6].valid := 1, [77].log_data[7].time := 3600.0, [77].log_data[7].valid := 1, [77].log_data[8].max := 1.0, [77].log_data[8].total := 3315.751, [77].log_data[8].time := 3600.0, [77].log_data[8].minminute := 55, [77].log_data[8].valid := 1, [77].log_data[9].max := 1.0, [77].log_data[9].total := 3315.751, [77].log_data[9].time := 3600.0, [77].log_data[9].minminute := 55, [77].log_data[9].valid := 1, [77].log_data[10].min := 1.0, [77].log_data[10].max := 1.0, [77].log_data[10].total := 3600.0, [77].log_data[10].time := 3600.0, [77].log_data[10].valid := 1, [77].log_data[11].time := 3600.0, [77].log_data[11].valid := 1, [77].log_data[12].min := 1.0, [77].log_data[12].max := 1.0, [77].log_data[12].total := 3600.0, [77].log_data[12].time := 3600.0, [77].log_data[12].valid := 1, [77].log_data[13].min := 1.0, [77].log_data[13].max := 1.0, [77].log_data[13].total := 3600.0, [77].log_data[13].time := 3600.0, [77].log_data[13].valid := 1, [77].log_data[14].time := 3600.0, [77].log_data[14].valid := 1, [77].log_data[15].time := 3600.0, [77].log_data[15].valid := 1, [77].log_data[16].time := 3600.0, [77].log_data[16].valid := 1, [77].log_data[17].min := 1.0,
        [77].log_data[17].max := 1.0, [77].log_data[17].total := 3600.0, [77].log_data[17].time := 3600.0, [77].log_data[17].valid := 1, [77].log_data[18].time := 3600.0, [77].log_data[18].valid := 1, [77].log_data[19].time := 3600.0, [77].log_data[19].valid := 1, [77].log_data[20].time := 3600.0, [77].log_data[20].valid := 1, [77].log_data[21].min := 1.0, [77].log_data[21].max := 1.0, [77].log_data[21].total := 3600.0, [77].log_data[21].time := 3600.0, [77].log_data[21].valid := 1, [77].log_data[22].time := 3600.0, [77].log_data[22].valid := 1, [77].log_data[23].time := 3600.0, [77].log_data[23].valid := 1, [77].log_data[24].time := 3600.0, [77].log_data[24].valid := 1, [77].log_data[25].time := 3600.0, [77].log_data[25].valid := 1, [77].log_data[26].time := 3600.0, [77].log_data[26].valid := 1, [77].log_data[27].time := 3600.0, [77].log_data[27].valid := 1, [77].log_data[28].time := 3600.0, [77].log_data[28].valid := 1, [77].log_data[29].min := 1.0, [77].log_data[29].max := 1.0, [77].log_data[29].total := 3600.0, [77].log_data[29].time := 3600.0, [77].log_data[29].valid := 1, [77].log_data[30].min := 1.0, [77].log_data[30].max := 1.0, [77].log_data[30].total := 3600.0, [77].log_data[30].time := 3600.0, [77].log_data[30].valid := 1, [77].log_data[31].max := 1.0, [77].log_data[31].total := 1575.2471, [77].log_data[31].time := 3600.0, [77].log_data[31].maxminute := 5, [77].log_data[31].valid := 1, [77].log_data[32].max := 1.0, [77].log_data[32].total := 1303.0, [77].log_data[32].time := 3600.0, [77].log_data[32].minminute := 3, [77].log_data[32].valid := 1, [77].log_data[33].time := 3600.0, [77].log_data[33].valid := 1, [77].log_data[34].time := 3600.0, [77].log_data[34].valid := 1, [77].log_data[35].max := 1.0, [77].log_data[35].total := 1328.2471, [77].log_data[35].time := 3600.0, [77].log_data[35].maxminute := 9, [77].log_data[35].valid := 1, [77].log_data[36].max := 1.0, [77].log_data[36].total := 1549.998,
        [77].log_data[36].time := 3600.0, [77].log_data[36].minminute := 7, [77].log_data[36].valid := 1, [77].log_data[37].time := 3600.0, [77].log_data[37].valid := 1, [77].log_data[38].time := 3600.0, [77].log_data[38].valid := 1, [77].log_data[39].min := 0.9956484, [77].log_data[39].max := 1.0080148, [77].log_data[39].total := 3607.7026, [77].log_data[39].time := 3600.0, [77].log_data[39].minminute := 44, [77].log_data[39].maxminute := 40, [77].log_data[39].valid := 1, [77].log_data[40].min := 7.5742097, [77].log_data[40].max := 7.609111, [77].log_data[40].total := 27335.467, [77].log_data[40].time := 3600.0, [77].log_data[40].minminute := 28, [77].log_data[40].maxminute := 24, [77].log_data[40].valid := 1, [77].log_data[41].min := 0.022540038, [77].log_data[41].max := 0.033139892, [77].log_data[41].total := 100.900345, [77].log_data[41].time := 3600.0, [77].log_data[41].minminute := 41, [77].log_data[41].maxminute := 16, [77].log_data[41].valid := 1, [77].log_data[42].min := 2.2916427, [77].log_data[42].max := 2.2963536, [77].log_data[42].total := 8259.254, [77].log_data[42].time := 3600.0, [77].log_data[42].minminute := 14, [77].log_data[42].maxminute := 39, [77].log_data[42].valid := 1, [77].log_data[43].min := -0.27999878, [77].log_data[43].max := -0.26000214, [77].log_data[43].total := -989.81494, [77].log_data[43].time := 3600.0, [77].log_data[43].valid := 1, [77].log_data[44].min := -0.3199997, [77].log_data[44].max := -0.30000305, [77].log_data[44].total := -1080.0961, [77].log_data[44].time := 3600.0, [77].log_data[44].minminute := 55, [77].log_data[44].valid := 1, [77].log_data[45].time := 3600.0, [77].log_data[45].valid := 1, [77].log_data[46].time := 3600.0, [77].log_data[46].valid := 1, [77].log_data[47].time := 3600.0, [77].log_data[47].valid := 1, [77].log_data[48].min := 6.5750084, [77].log_data[48].max := 6.8069463, [77].log_data[48].total := 24206.191, [77].log_data[48].time := 3600.0, [77].log_data[48].minminute := 7, [77].log_data[48].maxminute := 22, [77].log_data[48].valid := 1, [77].log_data[49].min := 7.0228796,
        [77].log_data[49].max := 9.625507, [77].log_data[49].total := 31341.023, [77].log_data[49].time := 3600.0, [77].log_data[49].minminute := 4, [77].log_data[49].maxminute := 55, [77].log_data[49].valid := 1, [77].log_data[50].min := 1.9997966, [77].log_data[50].max := 2.0896587, [77].log_data[50].total := 7360.13, [77].log_data[50].time := 3600.0, [77].log_data[50].minminute := 55, [77].log_data[50].maxminute := 59, [77].log_data[50].valid := 1, [77].log_data[51].time := 3600.0, [77].log_data[51].valid := 1, [77].log_data[52].min := -2.9000015, [77].log_data[52].max := 0.11999512, [77].log_data[52].total := -7380.3057, [77].log_data[52].time := 3600.0, [77].log_data[52].minminute := 5, [77].log_data[52].maxminute := 3, [77].log_data[52].valid := 1, [77].log_data[53].min := -2.4800034, [77].log_data[53].max := 0.27999878, [77].log_data[53].total := -6775.32, [77].log_data[53].time := 3600.0, [77].log_data[53].minminute := 10, [77].log_data[53].maxminute := 19, [77].log_data[53].valid := 1, [77].log_data[54].max := 0.532, [77].log_data[54].total := 1142.4111, [77].log_data[54].time := 3600.0, [77].log_data[54].minminute := 3, [77].log_data[54].maxminute := 5, [77].log_data[54].valid := 1, [77].log_data[55].max := 0.5265, [77].log_data[55].total := 1142.5466, [77].log_data[55].time := 3600.0, [77].log_data[55].minminute := 7, [77].log_data[55].maxminute := 19, [77].log_data[55].valid := 1, [77].log_data[56].min := 0.16008857, [77].log_data[56].max := 0.16048115, [77].log_data[56].total := 576.8243, [77].log_data[56].time := 3600.0, [77].log_data[56].maxminute := 29, [77].log_data[56].valid := 1, [77].log_data[57].min := 0.25375885, [77].log_data[57].max := 0.25619283, [77].log_data[57].total := 915.5109, [77].log_data[57].time := 3600.0, [77].log_data[57].minminute := 39, [77].log_data[57].valid := 1, [77].log_data[58].time := 3600.0, [77].log_data[58].valid := 1, [77].log_data[59].time := 3600.0, [77].log_data[59].valid := 1, [77].log_data[60].valid := 1, [77].log_data[61].valid := 1, [77].log_data[62].valid := 1,
        [77].log_data[63].valid := 1, [77].log_data[64].valid := 1, [77].log_data[65].valid := 1, [77].log_data[66].valid := 1, [77].log_data[67].valid := 1, [77].log_data[68].valid := 1, [77].log_data[69].valid := 1, [77].log_data[70].valid := 1, [77].log_data[71].valid := 1, [77].log_data[72].valid := 1, [77].log_data[73].valid := 1, [77].log_data[74].valid := 1, [77].log_data[75].valid := 1, [77].log_data[76].valid := 1, [77].log_data[77].valid := 1, [77].log_data[78].valid := 1, [77].log_data[79].valid := 1, [77].log_data[80].valid := 1, [77].log_data[81].valid := 1, [77].log_data[82].valid := 1, [77].log_data[83].valid := 1, [77].log_data[84].valid := 1, [77].log_data[85].valid := 1, [77].log_data[86].valid := 1, [77].log_data[87].valid := 1, [77].log_data[88].valid := 1, [77].log_data[89].valid := 1, [77].log_data[90].valid := 1, [77].log_data[91].valid := 1, [77].log_data[92].valid := 1, [77].log_data[93].valid := 1, [77].log_data[94].valid := 1, [77].log_data[95].valid := 1, [77].log_data[96].valid := 1, [77].log_data[97].valid := 1, [77].log_data[98].valid := 1, [77].log_data[99].valid := 1, [77].log_data[100].valid := 1, [77].log_data[101].valid := 1, [77].log_data[102].valid := 1, [77].log_data[103].valid := 1, [77].log_data[104].valid := 1, [77].log_data[105].valid := 1, [77].log_data[106].valid := 1, [77].log_data[107].valid := 1, [77].log_data[108].valid := 1, [77].log_data[109].valid := 1, [77].log_data[110].valid := 1, [77].log_data[111].valid := 1, [77].log_data[112].valid := 1, [77].log_data[113].valid := 1, [77].log_data[114].valid := 1, [77].log_data[115].valid := 1, [77].log_data[116].valid := 1, [77].log_data[117].valid := 1, [77].log_data[118].valid := 1, [77].log_data[119].valid := 1, [77].log_data[120].valid := 1, [77].log_data[121].valid := 1, [77].log_data[122].valid := 1,
        [77].log_data[123].valid := 1, [77].log_data[124].valid := 1, [77].time.Year := 2023, [77].time.Month := 1, [77].time.Day := 16, [77].time.Hour := 8, [77].time.Minute := 59, [77].time.Second := 59, [78].log_data[0].min := 1.0, [78].log_data[0].max := 1.0, [78].log_data[0].total := 3600.0, [78].log_data[0].time := 3600.0, [78].log_data[0].valid := 1, [78].log_data[1].max := 1.0, [78].log_data[1].total := 553.5, [78].log_data[1].time := 3600.0, [78].log_data[1].maxminute := 14, [78].log_data[1].valid := 1, [78].log_data[2].max := 1.0, [78].log_data[2].total := 550.0, [78].log_data[2].time := 3600.0, [78].log_data[2].maxminute := 14, [78].log_data[2].valid := 1, [78].log_data[3].time := 3600.0, [78].log_data[3].valid := 1, [78].log_data[4].time := 3600.0, [78].log_data[4].valid := 1, [78].log_data[5].max := 1.0, [78].log_data[5].total := 245.5, [78].log_data[5].time := 3600.0, [78].log_data[5].maxminute := 16, [78].log_data[5].valid := 1, [78].log_data[6].time := 3600.0, [78].log_data[6].valid := 1, [78].log_data[7].time := 3600.0, [78].log_data[7].valid := 1, [78].log_data[8].max := 1.0, [78].log_data[8].total := 2501.249, [78].log_data[8].time := 3600.0, [78].log_data[8].maxminute := 18, [78].log_data[8].valid := 1, [78].log_data[9].max := 1.0, [78].log_data[9].total := 2497.749, [78].log_data[9].time := 3600.0, [78].log_data[9].maxminute := 18, [78].log_data[9].valid := 1, [78].log_data[10].min := 1.0, [78].log_data[10].max := 1.0, [78].log_data[10].total := 3600.0, [78].log_data[10].time := 3600.0, [78].log_data[10].valid := 1, [78].log_data[11].time := 3600.0, [78].log_data[11].valid := 1, [78].log_data[12].min := 1.0, [78].log_data[12].max := 1.0, [78].log_data[12].total := 3600.0, [78].log_data[12].time := 3600.0, [78].log_data[12].valid := 1, [78].log_data[13].min := 1.0, [78].log_data[13].max := 1.0,
        [78].log_data[13].total := 3600.0, [78].log_data[13].time := 3600.0, [78].log_data[13].valid := 1, [78].log_data[14].time := 3600.0, [78].log_data[14].valid := 1, [78].log_data[15].time := 3600.0, [78].log_data[15].valid := 1, [78].log_data[16].time := 3600.0, [78].log_data[16].valid := 1, [78].log_data[17].min := 1.0, [78].log_data[17].max := 1.0, [78].log_data[17].total := 3600.0, [78].log_data[17].time := 3600.0, [78].log_data[17].valid := 1, [78].log_data[18].time := 3600.0, [78].log_data[18].valid := 1, [78].log_data[19].time := 3600.0, [78].log_data[19].valid := 1, [78].log_data[20].time := 3600.0, [78].log_data[20].valid := 1, [78].log_data[21].min := 1.0, [78].log_data[21].max := 1.0, [78].log_data[21].total := 3600.0, [78].log_data[21].time := 3600.0, [78].log_data[21].valid := 1, [78].log_data[22].time := 3600.0, [78].log_data[22].valid := 1, [78].log_data[23].time := 3600.0, [78].log_data[23].valid := 1, [78].log_data[24].time := 3600.0, [78].log_data[24].valid := 1, [78].log_data[25].time := 3600.0, [78].log_data[25].valid := 1, [78].log_data[26].time := 3600.0, [78].log_data[26].valid := 1, [78].log_data[27].time := 3600.0, [78].log_data[27].valid := 1, [78].log_data[28].time := 3600.0, [78].log_data[28].valid := 1, [78].log_data[29].min := 1.0, [78].log_data[29].max := 1.0, [78].log_data[29].total := 3600.0, [78].log_data[29].time := 3600.0, [78].log_data[29].valid := 1, [78].log_data[30].min := 1.0, [78].log_data[30].max := 1.0, [78].log_data[30].total := 3600.0, [78].log_data[30].time := 3600.0, [78].log_data[30].valid := 1, [78].log_data[31].max := 1.0, [78].log_data[31].total := 1086.498, [78].log_data[31].time := 3600.0, [78].log_data[31].maxminute := 20, [78].log_data[31].valid := 1, [78].log_data[32].max := 1.0, [78].log_data[32].total := 1054.747, [78].log_data[32].time := 3600.0, [78].log_data[32].maxminute := 18, [78].log_data[32].valid := 1, [78].log_data[33].time := 3600.0,
        [78].log_data[33].valid := 1, [78].log_data[34].time := 3600.0, [78].log_data[34].valid := 1, [78].log_data[35].max := 1.0, [78].log_data[35].total := 1086.498, [78].log_data[35].time := 3600.0, [78].log_data[35].maxminute := 24, [78].log_data[35].valid := 1, [78].log_data[36].max := 1.0, [78].log_data[36].total := 1051.247, [78].log_data[36].time := 3600.0, [78].log_data[36].maxminute := 18, [78].log_data[36].valid := 1, [78].log_data[37].max := 7.519464, [78].log_data[37].total := 3597.0972, [78].log_data[37].time := 3600.0, [78].log_data[37].maxminute := 15, [78].log_data[37].valid := 1, [78].log_data[38].time := 3600.0, [78].log_data[38].valid := 1, [78].log_data[39].min := 0.9956484, [78].log_data[39].max := 1.0213233, [78].log_data[39].total := 3609.4648, [78].log_data[39].time := 3600.0, [78].log_data[39].minminute := 11, [78].log_data[39].maxminute := 21, [78].log_data[39].valid := 1, [78].log_data[40].min := 7.5758586, [78].log_data[40].max := 7.6047144, [78].log_data[40].total := 27338.354, [78].log_data[40].time := 3600.0, [78].log_data[40].minminute := 54, [78].log_data[40].maxminute := 57, [78].log_data[40].valid := 1, [78].log_data[41].min := 0.022540038, [78].log_data[41].max := 0.033139892, [78].log_data[41].total := 90.45787, [78].log_data[41].time := 3600.0, [78].log_data[41].maxminute := 56, [78].log_data[41].valid := 1, [78].log_data[42].min := 2.2917604, [78].log_data[42].max := 2.296236, [78].log_data[42].total := 8258.983, [78].log_data[42].time := 3600.0, [78].log_data[42].minminute := 29, [78].log_data[42].maxminute := 14, [78].log_data[42].valid := 1, [78].log_data[43].min := -0.27999878, [78].log_data[43].max := -0.26000214, [78].log_data[43].total := -990.1451, [78].log_data[43].time := 3600.0, [78].log_data[43].valid := 1, [78].log_data[44].min := -0.30000305, [78].log_data[44].max := -0.30000305, [78].log_data[44].total := -1080.0911, [78].log_data[44].time := 3600.0, [78].log_data[44].valid := 1, [78].log_data[45].time := 3600.0, [78].log_data[45].valid := 1, [78].log_data[46].time := 3600.0,
        [78].log_data[46].valid := 1, [78].log_data[47].time := 3600.0, [78].log_data[47].valid := 1, [78].log_data[48].min := 6.573634, [78].log_data[48].max := 6.9465485, [78].log_data[48].total := 24184.244, [78].log_data[48].time := 3600.0, [78].log_data[48].minminute := 45, [78].log_data[48].maxminute := 23, [78].log_data[48].valid := 1, [78].log_data[49].min := 6.850733, [78].log_data[49].max := 9.648866, [78].log_data[49].total := 29618.93, [78].log_data[49].time := 3600.0, [78].log_data[49].minminute := 42, [78].log_data[49].maxminute := 13, [78].log_data[49].valid := 1, [78].log_data[50].min := 2.069755, [78].log_data[50].max := 2.150313, [78].log_data[50].total := 7555.0293, [78].log_data[50].time := 3600.0, [78].log_data[50].minminute := 21, [78].log_data[50].maxminute := 18, [78].log_data[50].valid := 1, [78].log_data[51].time := 3600.0, [78].log_data[51].valid := 1, [78].log_data[52].min := -4.1399994, [78].log_data[52].max := 0.11999512, [78].log_data[52].total := -6942.0503, [78].log_data[52].time := 3600.0, [78].log_data[52].minminute := 18, [78].log_data[52].maxminute := 19, [78].log_data[52].valid := 1, [78].log_data[53].min := -4.0, [78].log_data[53].max := 0.2400055, [78].log_data[53].total := -6424.6904, [78].log_data[53].time := 3600.0, [78].log_data[53].minminute := 18, [78].log_data[53].maxminute := 24, [78].log_data[53].valid := 1, [78].log_data[54].max := 0.565, [78].log_data[54].total := 846.684, [78].log_data[54].time := 3600.0, [78].log_data[54].maxminute := 41, [78].log_data[54].valid := 1, [78].log_data[55].max := 0.522, [78].log_data[55].total := 845.482, [78].log_data[55].time := 3600.0, [78].log_data[55].maxminute := 25, [78].log_data[55].valid := 1, [78].log_data[56].min := 0.16004932, [78].log_data[56].max := 0.16048115, [78].log_data[56].total := 576.78796, [78].log_data[56].time := 3600.0, [78].log_data[56].minminute := 9, [78].log_data[56].maxminute := 11, [78].log_data[56].valid := 1, [78].log_data[57].min := 0.2515996, [78].log_data[57].max := 0.25419068, [78].log_data[57].total := 912.66437,
        [78].log_data[57].time := 3600.0, [78].log_data[57].minminute := 55, [78].log_data[57].maxminute := 1, [78].log_data[57].valid := 1, [78].log_data[58].time := 3600.0, [78].log_data[58].valid := 1, [78].log_data[59].time := 3600.0, [78].log_data[59].valid := 1, [78].log_data[60].valid := 1, [78].log_data[61].valid := 1, [78].log_data[62].valid := 1, [78].log_data[63].valid := 1, [78].log_data[64].valid := 1, [78].log_data[65].valid := 1, [78].log_data[66].valid := 1, [78].log_data[67].valid := 1, [78].log_data[68].valid := 1, [78].log_data[69].valid := 1, [78].log_data[70].valid := 1, [78].log_data[71].valid := 1, [78].log_data[72].valid := 1, [78].log_data[73].valid := 1, [78].log_data[74].valid := 1, [78].log_data[75].valid := 1, [78].log_data[76].valid := 1, [78].log_data[77].valid := 1, [78].log_data[78].valid := 1, [78].log_data[79].valid := 1, [78].log_data[80].valid := 1, [78].log_data[81].valid := 1, [78].log_data[82].valid := 1, [78].log_data[83].valid := 1, [78].log_data[84].valid := 1, [78].log_data[85].valid := 1, [78].log_data[86].valid := 1, [78].log_data[87].valid := 1, [78].log_data[88].valid := 1, [78].log_data[89].valid := 1, [78].log_data[90].valid := 1, [78].log_data[91].valid := 1, [78].log_data[92].valid := 1, [78].log_data[93].valid := 1, [78].log_data[94].valid := 1, [78].log_data[95].valid := 1, [78].log_data[96].valid := 1, [78].log_data[97].valid := 1, [78].log_data[98].valid := 1, [78].log_data[99].valid := 1, [78].log_data[100].valid := 1, [78].log_data[101].valid := 1, [78].log_data[102].valid := 1, [78].log_data[103].valid := 1, [78].log_data[104].valid := 1, [78].log_data[105].valid := 1, [78].log_data[106].valid := 1, [78].log_data[107].valid := 1, [78].log_data[108].valid := 1, [78].log_data[109].valid := 1, [78].log_data[110].valid := 1, [78].log_data[111].valid := 1,
        [78].log_data[112].valid := 1, [78].log_data[113].valid := 1, [78].log_data[114].valid := 1, [78].log_data[115].valid := 1, [78].log_data[116].valid := 1, [78].log_data[117].valid := 1, [78].log_data[118].valid := 1, [78].log_data[119].valid := 1, [78].log_data[120].valid := 1, [78].log_data[121].valid := 1, [78].log_data[122].valid := 1, [78].log_data[123].valid := 1, [78].log_data[124].valid := 1, [78].time.Year := 2023, [78].time.Month := 1, [78].time.Day := 16, [78].time.Hour := 9, [78].time.Minute := 59, [78].time.Second := 59, [79].log_data[0].min := 1.0, [79].log_data[0].max := 1.0, [79].log_data[0].total := 3599.5, [79].log_data[0].time := 3599.5, [79].log_data[0].valid := 1, [79].log_data[1].max := 1.0, [79].log_data[1].total := 564.0, [79].log_data[1].time := 3599.5, [79].log_data[1].maxminute := 47, [79].log_data[1].valid := 1, [79].log_data[2].max := 1.0, [79].log_data[2].total := 560.5, [79].log_data[2].time := 3599.5, [79].log_data[2].maxminute := 47, [79].log_data[2].valid := 1, [79].log_data[3].time := 3599.5, [79].log_data[3].valid := 1, [79].log_data[4].time := 3599.5, [79].log_data[4].valid := 1, [79].log_data[5].max := 1.0, [79].log_data[5].total := 239.5, [79].log_data[5].time := 3599.5, [79].log_data[5].maxminute := 50, [79].log_data[5].valid := 1, [79].log_data[6].time := 3599.5, [79].log_data[6].valid := 1, [79].log_data[7].time := 3599.5, [79].log_data[7].valid := 1, [79].log_data[8].max := 1.0, [79].log_data[8].total := 3314.0, [79].log_data[8].time := 3599.5, [79].log_data[8].minminute := 49, [79].log_data[8].valid := 1, [79].log_data[9].max := 1.0, [79].log_data[9].total := 3307.0, [79].log_data[9].time := 3599.5, [79].log_data[9].minminute := 49, [79].log_data[9].valid := 1, [79].log_data[10].min := 1.0, [79].log_data[10].max := 1.0, [79].log_data[10].total := 3599.5,
        [79].log_data[10].time := 3599.5, [79].log_data[10].valid := 1, [79].log_data[11].time := 3599.5, [79].log_data[11].valid := 1, [79].log_data[12].min := 1.0, [79].log_data[12].max := 1.0, [79].log_data[12].total := 3599.5, [79].log_data[12].time := 3599.5, [79].log_data[12].valid := 1, [79].log_data[13].min := 1.0, [79].log_data[13].max := 1.0, [79].log_data[13].total := 3599.5, [79].log_data[13].time := 3599.5, [79].log_data[13].valid := 1, [79].log_data[14].time := 3599.5, [79].log_data[14].valid := 1, [79].log_data[15].time := 3599.5, [79].log_data[15].valid := 1, [79].log_data[16].time := 3599.5, [79].log_data[16].valid := 1, [79].log_data[17].min := 1.0, [79].log_data[17].max := 1.0, [79].log_data[17].total := 3599.5, [79].log_data[17].time := 3599.5, [79].log_data[17].valid := 1, [79].log_data[18].time := 3599.5, [79].log_data[18].valid := 1, [79].log_data[19].time := 3599.5, [79].log_data[19].valid := 1, [79].log_data[20].time := 3599.5, [79].log_data[20].valid := 1, [79].log_data[21].min := 1.0, [79].log_data[21].max := 1.0, [79].log_data[21].total := 3599.5, [79].log_data[21].time := 3599.5, [79].log_data[21].valid := 1, [79].log_data[22].time := 3599.5, [79].log_data[22].valid := 1, [79].log_data[23].time := 3599.5, [79].log_data[23].valid := 1, [79].log_data[24].time := 3599.5, [79].log_data[24].valid := 1, [79].log_data[25].time := 3599.5, [79].log_data[25].valid := 1, [79].log_data[26].time := 3599.5, [79].log_data[26].valid := 1, [79].log_data[27].time := 3599.5, [79].log_data[27].valid := 1, [79].log_data[28].time := 3599.5, [79].log_data[28].valid := 1, [79].log_data[29].min := 1.0, [79].log_data[29].max := 1.0, [79].log_data[29].total := 3599.5, [79].log_data[29].time := 3599.5, [79].log_data[29].valid := 1, [79].log_data[30].min := 1.0, [79].log_data[30].max := 1.0, [79].log_data[30].total := 3599.5, [79].log_data[30].time := 3599.5, [79].log_data[30].valid := 1,
        [79].log_data[31].max := 1.0, [79].log_data[31].total := 1375.7471, [79].log_data[31].time := 3599.5, [79].log_data[31].maxminute := 2, [79].log_data[31].valid := 1, [79].log_data[32].max := 1.0, [79].log_data[32].total := 1427.0, [79].log_data[32].time := 3599.5, [79].log_data[32].minminute := 1, [79].log_data[32].valid := 1, [79].log_data[33].time := 3599.5, [79].log_data[33].valid := 1, [79].log_data[34].time := 3599.5, [79].log_data[34].valid := 1, [79].log_data[35].max := 1.0, [79].log_data[35].total := 1125.7471, [79].log_data[35].time := 3599.5, [79].log_data[35].maxminute := 7, [79].log_data[35].valid := 1, [79].log_data[36].max := 1.0, [79].log_data[36].total := 1736.7471, [79].log_data[36].time := 3599.5, [79].log_data[36].minminute := 5, [79].log_data[36].valid := 1, [79].log_data[37].max := 7.2348413, [79].log_data[37].total := 3546.9075, [79].log_data[37].time := 3599.5, [79].log_data[37].maxminute := 48, [79].log_data[37].valid := 1, [79].log_data[38].time := 3599.5, [79].log_data[38].valid := 1, [79].log_data[39].min := 0.9951773, [79].log_data[39].max := 1.02097, [79].log_data[39].total := 3608.7307, [79].log_data[39].time := 3599.5, [79].log_data[39].minminute := 42, [79].log_data[39].maxminute := 54, [79].log_data[39].valid := 1, [79].log_data[40].min := 7.5687137, [79].log_data[40].max := 7.609111, [79].log_data[40].total := 27333.996, [79].log_data[40].time := 3599.5, [79].log_data[40].minminute := 34, [79].log_data[40].maxminute := 41, [79].log_data[40].valid := 1, [79].log_data[41].min := 0.02273633, [79].log_data[41].max := 0.03628052, [79].log_data[41].total := 102.158676, [79].log_data[41].time := 3599.5, [79].log_data[41].minminute := 23, [79].log_data[41].maxminute := 56, [79].log_data[41].valid := 1, [79].log_data[42].min := 2.2912893, [79].log_data[42].max := 2.2963536, [79].log_data[42].total := 8257.793, [79].log_data[42].time := 3599.5, [79].log_data[42].minminute := 13, [79].log_data[42].maxminute := 52, [79].log_data[42].valid := 1, [79].log_data[43].min := -0.27999878,
        [79].log_data[43].max := -0.26000214, [79].log_data[43].total := -965.21716, [79].log_data[43].time := 3599.5, [79].log_data[43].valid := 1, [79].log_data[44].min := -0.30000305, [79].log_data[44].max := -0.30000305, [79].log_data[44].total := -1079.941, [79].log_data[44].time := 3599.5, [79].log_data[44].valid := 1, [79].log_data[45].time := 3599.5, [79].log_data[45].valid := 1, [79].log_data[46].time := 3599.5, [79].log_data[46].valid := 1, [79].log_data[47].time := 3599.5, [79].log_data[47].valid := 1, [79].log_data[48].min := 6.739068, [79].log_data[48].max := 6.9663343, [79].log_data[48].total := 24376.168, [79].log_data[48].time := 3599.5, [79].log_data[48].minminute := 49, [79].log_data[48].maxminute := 56, [79].log_data[48].valid := 1, [79].log_data[49].min := 7.8685026, [79].log_data[49].max := 9.629629, [79].log_data[49].total := 33376.152, [79].log_data[49].time := 3599.5, [79].log_data[49].minminute := 59, [79].log_data[49].maxminute := 48, [79].log_data[49].valid := 1, [79].log_data[50].min := 1.9993255, [79].log_data[50].max := 2.151373, [79].log_data[50].total := 7387.153, [79].log_data[50].time := 3599.5, [79].log_data[50].minminute := 49, [79].log_data[50].maxminute := 54, [79].log_data[50].valid := 1, [79].log_data[51].time := 3599.5, [79].log_data[51].valid := 1, [79].log_data[52].min := -3.8399963, [79].log_data[52].max := 0.11999512, [79].log_data[52].total := -7226.2876, [79].log_data[52].time := 3599.5, [79].log_data[52].minminute := 54, [79].log_data[52].maxminute := 1, [79].log_data[52].valid := 1, [79].log_data[53].min := -3.9399948, [79].log_data[53].max := 0.22000122, [79].log_data[53].total := -6825.5684, [79].log_data[53].time := 3599.5, [79].log_data[53].minminute := 54, [79].log_data[53].maxminute := 16, [79].log_data[53].valid := 1, [79].log_data[54].max := 0.5405, [79].log_data[54].total := 1110.355, [79].log_data[54].time := 3599.5, [79].log_data[54].minminute := 1, [79].log_data[54].maxminute := 24, [79].log_data[54].valid := 1, [79].log_data[55].max := 0.5395, [79].log_data[55].total := 1134.2974,
        [79].log_data[55].time := 3599.5, [79].log_data[55].minminute := 5, [79].log_data[55].maxminute := 54, [79].log_data[55].valid := 1, [79].log_data[56].min := 0.15993154, [79].log_data[56].max := 0.16044189, [79].log_data[56].total := 576.51, [79].log_data[56].time := 3599.5, [79].log_data[56].minminute := 28, [79].log_data[56].maxminute := 33, [79].log_data[56].valid := 1, [79].log_data[57].min := 0.25156036, [79].log_data[57].max := 0.2520707, [79].log_data[57].total := 906.3389, [79].log_data[57].time := 3599.5, [79].log_data[57].minminute := 18, [79].log_data[57].maxminute := 23, [79].log_data[57].valid := 1, [79].log_data[58].time := 3599.5, [79].log_data[58].valid := 1, [79].log_data[59].time := 3599.5, [79].log_data[59].valid := 1, [79].log_data[60].valid := 1, [79].log_data[61].valid := 1, [79].log_data[62].valid := 1, [79].log_data[63].valid := 1, [79].log_data[64].valid := 1, [79].log_data[65].valid := 1, [79].log_data[66].valid := 1, [79].log_data[67].valid := 1, [79].log_data[68].valid := 1, [79].log_data[69].valid := 1, [79].log_data[70].valid := 1, [79].log_data[71].valid := 1, [79].log_data[72].valid := 1, [79].log_data[73].valid := 1, [79].log_data[74].valid := 1, [79].log_data[75].valid := 1, [79].log_data[76].valid := 1, [79].log_data[77].valid := 1, [79].log_data[78].valid := 1, [79].log_data[79].valid := 1, [79].log_data[80].valid := 1, [79].log_data[81].valid := 1, [79].log_data[82].valid := 1, [79].log_data[83].valid := 1, [79].log_data[84].valid := 1, [79].log_data[85].valid := 1, [79].log_data[86].valid := 1, [79].log_data[87].valid := 1, [79].log_data[88].valid := 1, [79].log_data[89].valid := 1, [79].log_data[90].valid := 1, [79].log_data[91].valid := 1, [79].log_data[92].valid := 1, [79].log_data[93].valid := 1, [79].log_data[94].valid := 1, [79].log_data[95].valid := 1, [79].log_data[96].valid := 1, [79].log_data[97].valid := 1,
        [79].log_data[98].valid := 1, [79].log_data[99].valid := 1, [79].log_data[100].valid := 1, [79].log_data[101].valid := 1, [79].log_data[102].valid := 1, [79].log_data[103].valid := 1, [79].log_data[104].valid := 1, [79].log_data[105].valid := 1, [79].log_data[106].valid := 1, [79].log_data[107].valid := 1, [79].log_data[108].valid := 1, [79].log_data[109].valid := 1, [79].log_data[110].valid := 1, [79].log_data[111].valid := 1, [79].log_data[112].valid := 1, [79].log_data[113].valid := 1, [79].log_data[114].valid := 1, [79].log_data[115].valid := 1, [79].log_data[116].valid := 1, [79].log_data[117].valid := 1, [79].log_data[118].valid := 1, [79].log_data[119].valid := 1, [79].log_data[120].valid := 1, [79].log_data[121].valid := 1, [79].log_data[122].valid := 1, [79].log_data[123].valid := 1, [79].log_data[124].valid := 1, [79].time.Year := 2023, [79].time.Month := 1, [79].time.Day := 16, [79].time.Hour := 10, [79].time.Minute := 59, [79].time.Second := 59, [80].log_data[0].min := 1.0, [80].log_data[0].max := 1.0, [80].log_data[0].total := 3600.0, [80].log_data[0].time := 3600.0, [80].log_data[0].valid := 1, [80].log_data[1].time := 3600.0, [80].log_data[1].valid := 1, [80].log_data[2].time := 3600.0, [80].log_data[2].valid := 1, [80].log_data[3].time := 3600.0, [80].log_data[3].valid := 1, [80].log_data[4].time := 3600.0, [80].log_data[4].valid := 1, [80].log_data[5].time := 3600.0, [80].log_data[5].valid := 1, [80].log_data[6].time := 3600.0, [80].log_data[6].valid := 1, [80].log_data[7].time := 3600.0, [80].log_data[7].valid := 1, [80].log_data[8].min := 1.0, [80].log_data[8].max := 1.0, [80].log_data[8].total := 3600.0, [80].log_data[8].time := 3600.0, [80].log_data[8].valid := 1, [80].log_data[9].min := 1.0, [80].log_data[9].max := 1.0, [80].log_data[9].total := 3600.0,
        [80].log_data[9].time := 3600.0, [80].log_data[9].valid := 1, [80].log_data[10].min := 1.0, [80].log_data[10].max := 1.0, [80].log_data[10].total := 3600.0, [80].log_data[10].time := 3600.0, [80].log_data[10].valid := 1, [80].log_data[11].time := 3600.0, [80].log_data[11].valid := 1, [80].log_data[12].min := 1.0, [80].log_data[12].max := 1.0, [80].log_data[12].total := 3600.0, [80].log_data[12].time := 3600.0, [80].log_data[12].valid := 1, [80].log_data[13].min := 1.0, [80].log_data[13].max := 1.0, [80].log_data[13].total := 3600.0, [80].log_data[13].time := 3600.0, [80].log_data[13].valid := 1, [80].log_data[14].time := 3600.0, [80].log_data[14].valid := 1, [80].log_data[15].time := 3600.0, [80].log_data[15].valid := 1, [80].log_data[16].time := 3600.0, [80].log_data[16].valid := 1, [80].log_data[17].min := 1.0, [80].log_data[17].max := 1.0, [80].log_data[17].total := 3600.0, [80].log_data[17].time := 3600.0, [80].log_data[17].valid := 1, [80].log_data[18].time := 3600.0, [80].log_data[18].valid := 1, [80].log_data[19].time := 3600.0, [80].log_data[19].valid := 1, [80].log_data[20].time := 3600.0, [80].log_data[20].valid := 1, [80].log_data[21].min := 1.0, [80].log_data[21].max := 1.0, [80].log_data[21].total := 3600.0, [80].log_data[21].time := 3600.0, [80].log_data[21].valid := 1, [80].log_data[22].time := 3600.0, [80].log_data[22].valid := 1, [80].log_data[23].time := 3600.0, [80].log_data[23].valid := 1, [80].log_data[24].time := 3600.0, [80].log_data[24].valid := 1, [80].log_data[25].time := 3600.0, [80].log_data[25].valid := 1, [80].log_data[26].time := 3600.0, [80].log_data[26].valid := 1, [80].log_data[27].time := 3600.0, [80].log_data[27].valid := 1, [80].log_data[28].time := 3600.0, [80].log_data[28].valid := 1, [80].log_data[29].min := 1.0, [80].log_data[29].max := 1.0, [80].log_data[29].total := 3600.0, [80].log_data[29].time := 3600.0, [80].log_data[29].valid := 1,
        [80].log_data[30].min := 1.0, [80].log_data[30].max := 1.0, [80].log_data[30].total := 3600.0, [80].log_data[30].time := 3600.0, [80].log_data[30].valid := 1, [80].log_data[31].max := 1.0, [80].log_data[31].total := 1629.7471, [80].log_data[31].time := 3600.0, [80].log_data[31].valid := 1, [80].log_data[32].max := 1.0, [80].log_data[32].total := 1504.2471, [80].log_data[32].time := 3600.0, [80].log_data[32].maxminute := 10, [80].log_data[32].valid := 1, [80].log_data[33].time := 3600.0, [80].log_data[33].valid := 1, [80].log_data[34].time := 3600.0, [80].log_data[34].valid := 1, [80].log_data[35].max := 1.0, [80].log_data[35].total := 1629.7471, [80].log_data[35].time := 3600.0, [80].log_data[35].maxminute := 4, [80].log_data[35].valid := 1, [80].log_data[36].max := 1.0, [80].log_data[36].total := 1440.7471, [80].log_data[36].time := 3600.0, [80].log_data[36].minminute := 3, [80].log_data[36].valid := 1, [80].log_data[37].time := 3600.0, [80].log_data[37].valid := 1, [80].log_data[38].time := 3600.0, [80].log_data[38].valid := 1, [80].log_data[39].min := 0.9960017, [80].log_data[39].max := 1.0074259, [80].log_data[39].total := 3604.5232, [80].log_data[39].time := 3600.0, [80].log_data[39].minminute := 15, [80].log_data[39].maxminute := 51, [80].log_data[39].valid := 1, [80].log_data[40].min := 7.5871253, [80].log_data[40].max := 7.5989423, [80].log_data[40].total := 27339.645, [80].log_data[40].time := 3600.0, [80].log_data[40].minminute := 30, [80].log_data[40].maxminute := 55, [80].log_data[40].valid := 1, [80].log_data[41].min := 0.023717772, [80].log_data[41].max := 0.03628052, [80].log_data[41].total := 111.446106, [80].log_data[41].time := 3600.0, [80].log_data[41].minminute := 15, [80].log_data[41].maxminute := 50, [80].log_data[41].valid := 1, [80].log_data[42].min := 2.2916427, [80].log_data[42].max := 2.2963536, [80].log_data[42].total := 8258.862, [80].log_data[42].time := 3600.0, [80].log_data[42].minminute := 40, [80].log_data[42].maxminute := 48, [80].log_data[42].valid := 1,
        [80].log_data[43].min := -0.27999878, [80].log_data[43].max := -0.26000214, [80].log_data[43].total := -968.2052, [80].log_data[43].time := 3600.0, [80].log_data[43].valid := 1, [80].log_data[44].min := -0.30000305, [80].log_data[44].max := -0.30000305, [80].log_data[44].total := -1080.0911, [80].log_data[44].time := 3600.0, [80].log_data[44].valid := 1, [80].log_data[45].time := 3600.0, [80].log_data[45].valid := 1, [80].log_data[46].time := 3600.0, [80].log_data[46].valid := 1, [80].log_data[47].time := 3600.0, [80].log_data[47].valid := 1, [80].log_data[48].min := 6.578031, [80].log_data[48].max := 6.8110685, [80].log_data[48].total := 24183.033, [80].log_data[48].time := 3600.0, [80].log_data[48].minminute := 18, [80].log_data[48].maxminute := 35, [80].log_data[48].valid := 1, [80].log_data[49].min := 6.7712345, [80].log_data[49].max := 9.523436, [80].log_data[49].total := 29130.377, [80].log_data[49].time := 3600.0, [80].log_data[49].minminute := 18, [80].log_data[49].maxminute := 59, [80].log_data[49].valid := 1, [80].log_data[50].min := 2.0317135, [80].log_data[50].max := 2.1148627, [80].log_data[50].total := 7472.842, [80].log_data[50].time := 3600.0, [80].log_data[50].minminute := 59, [80].log_data[50].valid := 1, [80].log_data[51].time := 3600.0, [80].log_data[51].valid := 1, [80].log_data[52].min := -3.0200043, [80].log_data[52].max := 0.11999512, [80].log_data[52].total := -7767.737, [80].log_data[52].time := 3600.0, [80].log_data[52].minminute := 21, [80].log_data[52].valid := 1, [80].log_data[53].min := -2.5600052, [80].log_data[53].max := 0.2400055, [80].log_data[53].total := -7008.7046, [80].log_data[53].time := 3600.0, [80].log_data[53].minminute := 15, [80].log_data[53].maxminute := 4, [80].log_data[53].valid := 1, [80].log_data[54].max := 0.5325, [80].log_data[54].total := 1241.9974, [80].log_data[54].time := 3600.0, [80].log_data[54].maxminute := 21, [80].log_data[54].valid := 1, [80].log_data[55].max := 0.5365, [80].log_data[55].total := 1217.1273, [80].log_data[55].time := 3600.0, [80].log_data[55].minminute := 3,
        [80].log_data[55].maxminute := 25, [80].log_data[55].valid := 1, [80].log_data[56].min := 0.15981378, [80].log_data[56].max := 0.16036338, [80].log_data[56].total := 576.21326, [80].log_data[56].time := 3600.0, [80].log_data[56].minminute := 29, [80].log_data[56].maxminute := 3, [80].log_data[56].valid := 1, [80].log_data[57].min := 0.24959746, [80].log_data[57].max := 0.2519922, [80].log_data[57].total := 901.7906, [80].log_data[57].time := 3600.0, [80].log_data[57].minminute := 31, [80].log_data[57].maxminute := 14, [80].log_data[57].valid := 1, [80].log_data[58].time := 3600.0, [80].log_data[58].valid := 1, [80].log_data[59].time := 3600.0, [80].log_data[59].valid := 1, [80].log_data[60].valid := 1, [80].log_data[61].valid := 1, [80].log_data[62].valid := 1, [80].log_data[63].valid := 1, [80].log_data[64].valid := 1, [80].log_data[65].valid := 1, [80].log_data[66].valid := 1, [80].log_data[67].valid := 1, [80].log_data[68].valid := 1, [80].log_data[69].valid := 1, [80].log_data[70].valid := 1, [80].log_data[71].valid := 1, [80].log_data[72].valid := 1, [80].log_data[73].valid := 1, [80].log_data[74].valid := 1, [80].log_data[75].valid := 1, [80].log_data[76].valid := 1, [80].log_data[77].valid := 1, [80].log_data[78].valid := 1, [80].log_data[79].valid := 1, [80].log_data[80].valid := 1, [80].log_data[81].valid := 1, [80].log_data[82].valid := 1, [80].log_data[83].valid := 1, [80].log_data[84].valid := 1, [80].log_data[85].valid := 1, [80].log_data[86].valid := 1, [80].log_data[87].valid := 1, [80].log_data[88].valid := 1, [80].log_data[89].valid := 1, [80].log_data[90].valid := 1, [80].log_data[91].valid := 1, [80].log_data[92].valid := 1, [80].log_data[93].valid := 1, [80].log_data[94].valid := 1, [80].log_data[95].valid := 1, [80].log_data[96].valid := 1, [80].log_data[97].valid := 1, [80].log_data[98].valid := 1, [80].log_data[99].valid := 1,
        [80].log_data[100].valid := 1, [80].log_data[101].valid := 1, [80].log_data[102].valid := 1, [80].log_data[103].valid := 1, [80].log_data[104].valid := 1, [80].log_data[105].valid := 1, [80].log_data[106].valid := 1, [80].log_data[107].valid := 1, [80].log_data[108].valid := 1, [80].log_data[109].valid := 1, [80].log_data[110].valid := 1, [80].log_data[111].valid := 1, [80].log_data[112].valid := 1, [80].log_data[113].valid := 1, [80].log_data[114].valid := 1, [80].log_data[115].valid := 1, [80].log_data[116].valid := 1, [80].log_data[117].valid := 1, [80].log_data[118].valid := 1, [80].log_data[119].valid := 1, [80].log_data[120].valid := 1, [80].log_data[121].valid := 1, [80].log_data[122].valid := 1, [80].log_data[123].valid := 1, [80].log_data[124].valid := 1, [80].time.Year := 2023, [80].time.Month := 1, [80].time.Day := 16, [80].time.Hour := 11, [80].time.Minute := 59, [80].time.Second := 59, [81].log_data[0].min := 1.0, [81].log_data[0].max := 1.0, [81].log_data[0].total := 3600.0, [81].log_data[0].time := 3600.0, [81].log_data[0].valid := 1, [81].log_data[1].max := 1.0, [81].log_data[1].total := 541.5, [81].log_data[1].time := 3600.0, [81].log_data[1].maxminute := 35, [81].log_data[1].valid := 1, [81].log_data[2].max := 1.0, [81].log_data[2].total := 538.0, [81].log_data[2].time := 3600.0, [81].log_data[2].maxminute := 35, [81].log_data[2].valid := 1, [81].log_data[3].time := 3600.0, [81].log_data[3].valid := 1, [81].log_data[4].time := 3600.0, [81].log_data[4].valid := 1, [81].log_data[5].max := 1.0, [81].log_data[5].total := 241.0, [81].log_data[5].time := 3600.0, [81].log_data[5].maxminute := 37, [81].log_data[5].valid := 1, [81].log_data[6].time := 3600.0, [81].log_data[6].valid := 1, [81].log_data[7].time := 3600.0, [81].log_data[7].valid := 1, [81].log_data[8].max := 1.0,
        [81].log_data[8].total := 2168.5, [81].log_data[8].time := 3600.0, [81].log_data[8].minminute := 15, [81].log_data[8].valid := 1, [81].log_data[9].max := 1.0, [81].log_data[9].total := 2165.0, [81].log_data[9].time := 3600.0, [81].log_data[9].minminute := 15, [81].log_data[9].valid := 1, [81].log_data[10].min := 1.0, [81].log_data[10].max := 1.0, [81].log_data[10].total := 3600.0, [81].log_data[10].time := 3600.0, [81].log_data[10].valid := 1, [81].log_data[11].time := 3600.0, [81].log_data[11].valid := 1, [81].log_data[12].min := 1.0, [81].log_data[12].max := 1.0, [81].log_data[12].total := 3600.0, [81].log_data[12].time := 3600.0, [81].log_data[12].valid := 1, [81].log_data[13].min := 1.0, [81].log_data[13].max := 1.0, [81].log_data[13].total := 3600.0, [81].log_data[13].time := 3600.0, [81].log_data[13].valid := 1, [81].log_data[14].time := 3600.0, [81].log_data[14].valid := 1, [81].log_data[15].time := 3600.0, [81].log_data[15].valid := 1, [81].log_data[16].time := 3600.0, [81].log_data[16].valid := 1, [81].log_data[17].min := 1.0, [81].log_data[17].max := 1.0, [81].log_data[17].total := 3600.0, [81].log_data[17].time := 3600.0, [81].log_data[17].valid := 1, [81].log_data[18].time := 3600.0, [81].log_data[18].valid := 1, [81].log_data[19].time := 3600.0, [81].log_data[19].valid := 1, [81].log_data[20].time := 3600.0, [81].log_data[20].valid := 1, [81].log_data[21].min := 1.0, [81].log_data[21].max := 1.0, [81].log_data[21].total := 3600.0, [81].log_data[21].time := 3600.0, [81].log_data[21].valid := 1, [81].log_data[22].time := 3600.0, [81].log_data[22].valid := 1, [81].log_data[23].time := 3600.0, [81].log_data[23].valid := 1, [81].log_data[24].time := 3600.0, [81].log_data[24].valid := 1, [81].log_data[25].time := 3600.0, [81].log_data[25].valid := 1, [81].log_data[26].time := 3600.0, [81].log_data[26].valid := 1, [81].log_data[27].time := 3600.0, [81].log_data[27].valid := 1,
        [81].log_data[28].time := 3600.0, [81].log_data[28].valid := 1, [81].log_data[29].min := 1.0, [81].log_data[29].max := 1.0, [81].log_data[29].total := 3600.0, [81].log_data[29].time := 3600.0, [81].log_data[29].valid := 1, [81].log_data[30].min := 1.0, [81].log_data[30].max := 1.0, [81].log_data[30].total := 3600.0, [81].log_data[30].time := 3600.0, [81].log_data[30].valid := 1, [81].log_data[31].max := 1.0, [81].log_data[31].total := 1075.7471, [81].log_data[31].time := 3600.0, [81].log_data[31].maxminute := 3, [81].log_data[31].valid := 1, [81].log_data[32].max := 1.0, [81].log_data[32].total := 737.0, [81].log_data[32].time := 3600.0, [81].log_data[32].minminute := 2, [81].log_data[32].valid := 1, [81].log_data[33].time := 3600.0, [81].log_data[33].valid := 1, [81].log_data[34].time := 3600.0, [81].log_data[34].valid := 1, [81].log_data[35].max := 1.0, [81].log_data[35].total := 988.998, [81].log_data[35].time := 3600.0, [81].log_data[35].maxminute := 7, [81].log_data[35].valid := 1, [81].log_data[36].max := 1.0, [81].log_data[36].total := 907.998, [81].log_data[36].time := 3600.0, [81].log_data[36].minminute := 6, [81].log_data[36].valid := 1, [81].log_data[37].max := 7.5359526, [81].log_data[37].total := 3519.987, [81].log_data[37].time := 3600.0, [81].log_data[37].maxminute := 36, [81].log_data[37].valid := 1, [81].log_data[38].time := 3600.0, [81].log_data[38].valid := 1, [81].log_data[39].min := 0.99529505, [81].log_data[39].max := 1.0216767, [81].log_data[39].total := 3608.1604, [81].log_data[39].time := 3600.0, [81].log_data[39].minminute := 17, [81].log_data[39].maxminute := 42, [81].log_data[39].valid := 1, [81].log_data[40].min := 7.5816298, [81].log_data[40].max := 7.603614, [81].log_data[40].total := 27338.26, [81].log_data[40].time := 3600.0, [81].log_data[40].minminute := 50, [81].log_data[40].maxminute := 42, [81].log_data[40].valid := 1, [81].log_data[41].min := 0.02273633, [81].log_data[41].max := 0.034317628, [81].log_data[41].total := 92.31216,
        [81].log_data[41].time := 3600.0, [81].log_data[41].minminute := 29, [81].log_data[41].maxminute := 3, [81].log_data[41].valid := 1, [81].log_data[42].min := 2.2916427, [81].log_data[42].max := 2.2964714, [81].log_data[42].total := 8258.903, [81].log_data[42].time := 3600.0, [81].log_data[42].minminute := 52, [81].log_data[42].maxminute := 31, [81].log_data[42].valid := 1, [81].log_data[43].min := -0.27999878, [81].log_data[43].max := -0.26000214, [81].log_data[43].total := -1001.1685, [81].log_data[43].time := 3600.0, [81].log_data[43].valid := 1, [81].log_data[44].min := -0.3199997, [81].log_data[44].max := -0.30000305, [81].log_data[44].total := -1081.622, [81].log_data[44].time := 3600.0, [81].log_data[44].minminute := 14, [81].log_data[44].valid := 1, [81].log_data[45].time := 3600.0, [81].log_data[45].valid := 1, [81].log_data[46].time := 3600.0, [81].log_data[46].valid := 1, [81].log_data[47].time := 3600.0, [81].log_data[47].valid := 1, [81].log_data[48].min := 6.645359, [81].log_data[48].max := 6.9292355, [81].log_data[48].total := 24350.293, [81].log_data[48].time := 3600.0, [81].log_data[48].minminute := 59, [81].log_data[48].maxminute := 40, [81].log_data[48].valid := 1, [81].log_data[49].min := 6.8984313, [81].log_data[49].max := 9.602541, [81].log_data[49].total := 32337.62, [81].log_data[49].time := 3600.0, [81].log_data[49].minminute := 59, [81].log_data[49].maxminute := 19, [81].log_data[49].valid := 1, [81].log_data[50].min := 1.9990901, [81].log_data[50].max := 2.150313, [81].log_data[50].total := 7512.422, [81].log_data[50].time := 3600.0, [81].log_data[50].minminute := 15, [81].log_data[50].maxminute := 39, [81].log_data[50].valid := 1, [81].log_data[51].time := 3600.0, [81].log_data[51].valid := 1, [81].log_data[52].min := -4.239998, [81].log_data[52].max := 0.11999512, [81].log_data[52].total := -6451.244, [81].log_data[52].time := 3600.0, [81].log_data[52].minminute := 39, [81].log_data[52].maxminute := 2, [81].log_data[52].valid := 1, [81].log_data[53].min := -3.9399948, [81].log_data[53].max := 0.27999878,
        [81].log_data[53].total := -6193.644, [81].log_data[53].time := 3600.0, [81].log_data[53].minminute := 39, [81].log_data[53].maxminute := 52, [81].log_data[53].valid := 1, [81].log_data[54].max := 0.5395, [81].log_data[54].total := 716.2571, [81].log_data[54].time := 3600.0, [81].log_data[54].minminute := 2, [81].log_data[54].maxminute := 48, [81].log_data[54].valid := 1, [81].log_data[55].max := 0.5465, [81].log_data[55].total := 751.527, [81].log_data[55].time := 3600.0, [81].log_data[55].minminute := 6, [81].log_data[55].maxminute := 42, [81].log_data[55].valid := 1, [81].log_data[56].min := 0.15981378, [81].log_data[56].max := 0.16024561, [81].log_data[56].total := 576.057, [81].log_data[56].time := 3600.0, [81].log_data[56].minminute := 58, [81].log_data[56].maxminute := 17, [81].log_data[56].valid := 1, [81].log_data[57].min := 0.24959746, [81].log_data[57].max := 0.25006855, [81].log_data[57].total := 899.22064, [81].log_data[57].time := 3600.0, [81].log_data[57].minminute := 17, [81].log_data[57].maxminute := 2, [81].log_data[57].valid := 1, [81].log_data[58].time := 3600.0, [81].log_data[58].valid := 1, [81].log_data[59].time := 3600.0, [81].log_data[59].valid := 1, [81].log_data[60].valid := 1, [81].log_data[61].valid := 1, [81].log_data[62].valid := 1, [81].log_data[63].valid := 1, [81].log_data[64].valid := 1, [81].log_data[65].valid := 1, [81].log_data[66].valid := 1, [81].log_data[67].valid := 1, [81].log_data[68].valid := 1, [81].log_data[69].valid := 1, [81].log_data[70].valid := 1, [81].log_data[71].valid := 1, [81].log_data[72].valid := 1, [81].log_data[73].valid := 1, [81].log_data[74].valid := 1, [81].log_data[75].valid := 1, [81].log_data[76].valid := 1, [81].log_data[77].valid := 1, [81].log_data[78].valid := 1, [81].log_data[79].valid := 1, [81].log_data[80].valid := 1, [81].log_data[81].valid := 1, [81].log_data[82].valid := 1, [81].log_data[83].valid := 1, [81].log_data[84].valid := 1,
        [81].log_data[85].valid := 1, [81].log_data[86].valid := 1, [81].log_data[87].valid := 1, [81].log_data[88].valid := 1, [81].log_data[89].valid := 1, [81].log_data[90].valid := 1, [81].log_data[91].valid := 1, [81].log_data[92].valid := 1, [81].log_data[93].valid := 1, [81].log_data[94].valid := 1, [81].log_data[95].valid := 1, [81].log_data[96].valid := 1, [81].log_data[97].valid := 1, [81].log_data[98].valid := 1, [81].log_data[99].valid := 1, [81].log_data[100].valid := 1, [81].log_data[101].valid := 1, [81].log_data[102].valid := 1, [81].log_data[103].valid := 1, [81].log_data[104].valid := 1, [81].log_data[105].valid := 1, [81].log_data[106].valid := 1, [81].log_data[107].valid := 1, [81].log_data[108].valid := 1, [81].log_data[109].valid := 1, [81].log_data[110].valid := 1, [81].log_data[111].valid := 1, [81].log_data[112].valid := 1, [81].log_data[113].valid := 1, [81].log_data[114].valid := 1, [81].log_data[115].valid := 1, [81].log_data[116].valid := 1, [81].log_data[117].valid := 1, [81].log_data[118].valid := 1, [81].log_data[119].valid := 1, [81].log_data[120].valid := 1, [81].log_data[121].valid := 1, [81].log_data[122].valid := 1, [81].log_data[123].valid := 1, [81].log_data[124].valid := 1, [81].time.Year := 2023, [81].time.Month := 1, [81].time.Day := 16, [81].time.Hour := 12, [81].time.Minute := 59, [81].time.Second := 59, [82].log_data[0].min := 1.0, [82].log_data[0].max := 1.0, [82].log_data[0].total := 3600.0, [82].log_data[0].time := 3600.0, [82].log_data[0].valid := 1, [82].log_data[1].time := 3600.0, [82].log_data[1].valid := 1, [82].log_data[2].time := 3600.0, [82].log_data[2].valid := 1, [82].log_data[3].time := 3600.0, [82].log_data[3].valid := 1, [82].log_data[4].time := 3600.0, [82].log_data[4].valid := 1, [82].log_data[5].time := 3600.0,
        [82].log_data[5].valid := 1, [82].log_data[6].time := 3600.0, [82].log_data[6].valid := 1, [82].log_data[7].time := 3600.0, [82].log_data[7].valid := 1, [82].log_data[8].min := 1.0, [82].log_data[8].max := 1.0, [82].log_data[8].total := 3600.0, [82].log_data[8].time := 3600.0, [82].log_data[8].valid := 1, [82].log_data[9].min := 1.0, [82].log_data[9].max := 1.0, [82].log_data[9].total := 3600.0, [82].log_data[9].time := 3600.0, [82].log_data[9].valid := 1, [82].log_data[10].min := 1.0, [82].log_data[10].max := 1.0, [82].log_data[10].total := 3600.0, [82].log_data[10].time := 3600.0, [82].log_data[10].valid := 1, [82].log_data[11].time := 3600.0, [82].log_data[11].valid := 1, [82].log_data[12].min := 1.0, [82].log_data[12].max := 1.0, [82].log_data[12].total := 3600.0, [82].log_data[12].time := 3600.0, [82].log_data[12].valid := 1, [82].log_data[13].min := 1.0, [82].log_data[13].max := 1.0, [82].log_data[13].total := 3600.0, [82].log_data[13].time := 3600.0, [82].log_data[13].valid := 1, [82].log_data[14].time := 3600.0, [82].log_data[14].valid := 1, [82].log_data[15].time := 3600.0, [82].log_data[15].valid := 1, [82].log_data[16].time := 3600.0, [82].log_data[16].valid := 1, [82].log_data[17].min := 1.0, [82].log_data[17].max := 1.0, [82].log_data[17].total := 3600.0, [82].log_data[17].time := 3600.0, [82].log_data[17].valid := 1, [82].log_data[18].time := 3600.0, [82].log_data[18].valid := 1, [82].log_data[19].time := 3600.0, [82].log_data[19].valid := 1, [82].log_data[20].time := 3600.0, [82].log_data[20].valid := 1, [82].log_data[21].min := 1.0, [82].log_data[21].max := 1.0, [82].log_data[21].total := 3600.0, [82].log_data[21].time := 3600.0, [82].log_data[21].valid := 1, [82].log_data[22].time := 3600.0, [82].log_data[22].valid := 1, [82].log_data[23].time := 3600.0, [82].log_data[23].valid := 1, [82].log_data[24].time := 3600.0, [82].log_data[24].valid := 1,
        [82].log_data[25].time := 3600.0, [82].log_data[25].valid := 1, [82].log_data[26].time := 3600.0, [82].log_data[26].valid := 1, [82].log_data[27].time := 3600.0, [82].log_data[27].valid := 1, [82].log_data[28].time := 3600.0, [82].log_data[28].valid := 1, [82].log_data[29].min := 1.0, [82].log_data[29].max := 1.0, [82].log_data[29].total := 3600.0, [82].log_data[29].time := 3600.0, [82].log_data[29].valid := 1, [82].log_data[30].min := 1.0, [82].log_data[30].max := 1.0, [82].log_data[30].total := 3600.0, [82].log_data[30].time := 3600.0, [82].log_data[30].valid := 1, [82].log_data[31].max := 1.0, [82].log_data[31].total := 1572.498, [82].log_data[31].time := 3600.0, [82].log_data[31].minminute := 8, [82].log_data[31].valid := 1, [82].log_data[32].max := 1.0, [82].log_data[32].total := 1586.2471, [82].log_data[32].time := 3600.0, [82].log_data[32].maxminute := 9, [82].log_data[32].valid := 1, [82].log_data[33].time := 3600.0, [82].log_data[33].valid := 1, [82].log_data[34].time := 3600.0, [82].log_data[34].valid := 1, [82].log_data[35].max := 1.0, [82].log_data[35].total := 1629.7471, [82].log_data[35].time := 3600.0, [82].log_data[35].maxminute := 3, [82].log_data[35].valid := 1, [82].log_data[36].max := 1.0, [82].log_data[36].total := 1440.998, [82].log_data[36].time := 3600.0, [82].log_data[36].minminute := 1, [82].log_data[36].valid := 1, [82].log_data[37].time := 3600.0, [82].log_data[37].valid := 1, [82].log_data[38].time := 3600.0, [82].log_data[38].valid := 1, [82].log_data[39].min := 0.9947063, [82].log_data[39].max := 1.004717, [82].log_data[39].total := 3601.0654, [82].log_data[39].time := 3600.0, [82].log_data[39].minminute := 52, [82].log_data[39].maxminute := 16, [82].log_data[39].valid := 1, [82].log_data[40].min := 7.58905, [82].log_data[40].max := 7.6019654, [82].log_data[40].total := 27341.656, [82].log_data[40].time := 3600.0, [82].log_data[40].minminute := 11, [82].log_data[40].maxminute := 1, [82].log_data[40].valid := 1,
        [82].log_data[41].min := 0.02273633, [82].log_data[41].max := 0.023325196, [82].log_data[41].total := 82.90513, [82].log_data[41].time := 3600.0, [82].log_data[41].maxminute := 18, [82].log_data[41].valid := 1, [82].log_data[42].min := 2.2907004, [82].log_data[42].max := 2.2964714, [82].log_data[42].total := 8259.012, [82].log_data[42].time := 3600.0, [82].log_data[42].minminute := 51, [82].log_data[42].maxminute := 21, [82].log_data[42].valid := 1, [82].log_data[43].min := -0.27999878, [82].log_data[43].max := -0.26000214, [82].log_data[43].total := -1007.3838, [82].log_data[43].time := 3600.0, [82].log_data[43].valid := 1, [82].log_data[44].min := -0.3199997, [82].log_data[44].max := -0.30000305, [82].log_data[44].total := -1117.9546, [82].log_data[44].time := 3600.0, [82].log_data[44].valid := 1, [82].log_data[45].time := 3600.0, [82].log_data[45].valid := 1, [82].log_data[46].time := 3600.0, [82].log_data[46].valid := 1, [82].log_data[47].time := 3600.0, [82].log_data[47].valid := 1, [82].log_data[48].min := 6.57968, [82].log_data[48].max := 6.7940297, [82].log_data[48].total := 24210.664, [82].log_data[48].time := 3600.0, [82].log_data[48].minminute := 8, [82].log_data[48].maxminute := 21, [82].log_data[48].valid := 1, [82].log_data[49].min := 6.805978, [82].log_data[49].max := 9.591352, [82].log_data[49].total := 30848.684, [82].log_data[49].time := 3600.0, [82].log_data[49].minminute := 3, [82].log_data[49].maxminute := 57, [82].log_data[49].valid := 1, [82].log_data[50].min := 2.0144007, [82].log_data[50].max := 2.1099162, [82].log_data[50].total := 7422.4824, [82].log_data[50].time := 3600.0, [82].log_data[50].minminute := 59, [82].log_data[50].valid := 1, [82].log_data[51].time := 3600.0, [82].log_data[51].valid := 1, [82].log_data[52].min := -2.7799988, [82].log_data[52].max := 0.11999512, [82].log_data[52].total := -7783.198, [82].log_data[52].time := 3600.0, [82].log_data[52].minminute := 20, [82].log_data[52].maxminute := 8, [82].log_data[52].valid := 1, [82].log_data[53].min := -2.4800034, [82].log_data[53].max := 0.27999878,
